# B&R Automation Studio project TD52 (part 50)

#### perm_par.var
```iecst
VAR
	tParaIntern : ParaHandler_typ; (*Connector type to perm_par*)
	tMM2ParaBase_ReadBack : MM2ParaBase_type; (*INTERNAL! V4.06 new readback structure for information from previous tasks*)
	bWriteDataObj : BOOL; (* TRUE=write data object module *)
	bDataObjLenErr : BOOL; (*Error occured in permem: data module size missmatch*)
	bCreateDataObj : BOOL; (* TRUE=create new data object *)
	bWriteOnce : BOOL; (* write permanent memory once *)
	DatObjCreate_01 : DatObjCreate; (* data object create *)
	DatObjInfoBak_02 : DatObjInfo; (* data object info *)
	DatObjDelete_01 : DatObjDelete; (* data object delete *)
	DatObjRead_01 : DatObjRead; (* data object read *)
	DatObjRead_02 : DatObjRead; (* manual initiated data object read *)
	DatObjWrite_01 : DatObjWrite; (* data object write *)
	DatObjDelete_02 : DatObjDelete; (* data object delete *)
	DatObjDelete_11 : DatObjDelete; (*Delete Backup File*)
	DatObjInfo_01 : DatObjInfo; (* data object info *)
	DatObjInfo_02 : DatObjInfo; (* data object info *)
	szModuleName : STRING[35]; (* module name of object *)
	szModuleNameBackup : STRING[35]; (* module name of posiibly created backup object *)
	DatObjCopy_01 : DatObjCopy;
	bCopyDataObj : BOOL;
	TON_WarnDelay : TON;
	TON_WritePMEM : TON; (* delay write permanent memory *)
	ulPMPointer : UDINT; (* adress of actual checksum value *)
	ulChecksum : UDINT; (* parameter checksum value *)
	pm_len : UDINT; (* permanent value lenght *)
	ulChecksumOld : UDINT; (* last vlaue of parameter checksum *)
	ulChkValue : UDINT; (* actual value of parameter pointer *)
	pm_id : UDINT; (* permanent value identifier *)
	pm_p : UDINT; (* permanent value pointer *)
	DatObjInfo_META : DatObjInfo;
	DatObjRead_META : DatObjRead;
	szMetaDataRaw : STRING[2000];
	szMetaData : ARRAY[0..4] OF STRING[35];
	szMetaDataVis : ARRAY[0..3] OF STRING[35];
	ssIndex : INT;
	ssCount : INT;
	ucMetaDataRaw : ARRAY[0..2000] OF USINT;
	ssCount2 : INT;
	szMetaDataFile : STRING[10];
	szText1 : STRING[20];
	pv_adr_IN_XX_tPB2MM : UDINT;
	pv_lng : UDINT;
	pv_lng_IN_XX_tPB2MM : UDINT;
	pv_lng_OUT_XX_tPB2MM : UDINT;
	szText2 : STRING[20];
	pv_adr_OUT_XX_tXX2PB : UDINT;
END_VAR
VAR CONSTANT
	ERR_NOERROR : UINT := 0;
END_VAR
VAR
	usPMWriteCnt : UINT;
	pm_Error : UDINT; (* permanent value error *) (* Deleted: pm : ParaMem_typ; permanent memory tags mathias, 22.8.11*)
	fun_Error : UDINT := 0; (*state > 0 = function error*)
	xLocalParaCheck : ParaCheckFUB; (*local function instance to check parameter values*)
	TON_ParaSetupOk : TON;
	bParaCheckSystemOk : BOOL;
	iDebug_ParaOkChecked : UDINT;
	bRestoreBackupDataObj : BOOL := FALSE;
	bRestoreDataObjContent : BOOL := FALSE;
	pm_id_backup : UDINT;
	pm_p_Backup : UDINT;
	DatObjCopy_02 : DatObjCopy;
	bDeleteBackupDataObj : BOOL := FALSE; (*Command to delete backup data module file on purpose*)
	bDebugPara : ARRAY[0..5] OF BOOL;
	ssIndex2 : INT;
	ssIndex3 : INT;
	ssIndex4 : INT;
	ssIndexVis : INT;
	szText : STRING[40];
	pv_adr_Para : UDINT;
	szParaSnippet : ARRAY[0..5] OF STRING[150];
	szParaIndex : STRING[10];
	slValue : DINT;
	iModuleDLD_ResetCount : INT;
	bDownloadDetected : BOOL;
	bFlagParaStructCopyWorking : BOOL; (*true, if cyclic para copying is active, 1 false cycle at every copy *)
	bStoreInitParaInDataObj : BOOL := FALSE;
	bTestflag : BOOL;
	bReadOutMETA_Once : BOOL;
	tParaCheck_iPvAdress : ARRAY[0..5] OF UDINT;
	tParaCheck_iPvLengt : ARRAY[0..5] OF UDINT;
	tParaCheck_rPvValue : ARRAY[0..5] OF REAL;
	tParaCheck_rRangeMIN : ARRAY[0..5] OF REAL;
	tParaCheck_rRangeMAX : ARRAY[0..5] OF REAL;
	tParaCheck_szPvName : ARRAY[0..5] OF STRING[35];
	ssFormatDetected : INT;
	szMetaDataPart : STRING[150];
	szFullTaskName : STRING[35];
	szFullMetaModuleName : STRING[35];
	debugLen : INT;
	debugSize : INT := 0;
	strcat_adr1 : UDINT;
	strcat_adr2 : UDINT;
	ssIndexTN : INT;
	bAlternate : BOOL;
	n : INT;
	iAlternateChecksum : DINT;
	iAlternateChecksumOld : DINT;
	ulDebugChkValue : ARRAY[0..999] OF UDINT;
	Adr1 : UDINT;
	Adr2 : UDINT;
	usPMWriteCntStepsize : UINT := 1; (*different step sizes to help debug*)
	usPMWriteCntXOR : UINT;
	usPMWriteCntAltSum : UINT;
	ulAdrPM : UDINT;
	usChkValuePM : USINT;
	ulAdrPara : UDINT;
	ulPara_len : UDINT;
	usChkValuePara : USINT;
	iDebugCountPMDifferences : DINT := 0;
	bEngineRunDetected : BOOL; (*detection status bit autocommand 100 /101  for engine run state*)
	ucMetaDataDebugInfoLine : ARRAY[0..24] OF STRING[80];
	ssIndexMand : INT := 0;
	szMetaDataMand : STRING[35];
	iMyErrorInfo_Autoreset : DINT; (*internal autoreset counter*)
	ssIndex_Version : INT; (*internal*)
	ssIndex_BU : INT; (*internal*)
	ssIndex_BU2 : INT; (*internal*)
END_VAR
```

### Program Logical/Customized/Cust_Internals/par_UniFile (IEC, version 0.99.0) - + obsolete

- par_UniFile.st (not readable text: treated as protected, skipped)

### Program Logical/Customized/Cust_Internals/par_UniString (IEC, version 1.06.0) - + obsolete

- par_UniString.st (not readable text: treated as protected, skipped)

### Program Logical/Customized/Cust_Internals/par_Universal_IO (IEC, version 1.16.0) - + obsolete

- par_Universal_IO.st (not readable text: treated as protected, skipped)

### Program Logical/Customized/Cust_Internals/MsgCUInternal (IEC, version 4.10.0) - + unchangeable module messages

- MsgCUInterCyclic.st (not readable text: treated as protected, skipped)

- MsgCUInterInit.st (not readable text: treated as protected, skipped)

#### MsgCUInter.var - Local variables
```iecst
(********************************************************************
 * COPYRIGHT -- INNIO Company
 ********************************************************************
 * Program: MsgCUInter
 * File: MsgCUInter.var
 * Author: zengerer
 * Created: September 10, 2013
 ********************************************************************
 * Local variables of program MsgCU
 ********************************************************************)
VAR
	iAdrAmmBase2MM : UDINT;
	iAdrMM2AmmBase : UDINT;
	xMsg13 : ARRAY[0..99] OF Msg; (*Array of Msg for Reserve Analog IN*)
	xMsg14 : ARRAY[0..99] OF Msg; (*Array of Msg for Reserve Analog IN*)
	xMsg1500 : Msg; (*Msg 1500 for Reserve Analog IN*)
	xMsg37 : ARRAY[0..99] OF Msg; (*Array of Msg for Reserve Analog IN*)
	xMsg38 : ARRAY[0..99] OF Msg; (*Array of Msg for Reserve Analog IN*)
	xMsg39 : ARRAY[0..99] OF Msg; (*Array of Msg for Reserve Analog IN*)
	xMsg89 : ARRAY[66..99] OF Msg; (*Array of Msg for CustomerIO and Reserve AI*)
END_VAR
```

### Program Logical/Customized/Cust_Internals/ran_Internal (IEC, version 4.12.0) - + processing of spare analog inputs,..

- ran_InternalCyclic.st (not readable text: treated as protected, skipped)

#### ran_Internal.var
```iecst
VAR
	xTON_lim_LoLo : ARRAY[0..120] OF TON;
	xTON_lim_lo : ARRAY[0..120] OF TON;
	xTON_lim_hi : ARRAY[0..120] OF TON;
	xTON_lim_HiHi : ARRAY[0..120] OF TON;
	xLCRScal_10 : LCRScal;
	xLCRScal_15 : LCRScal;
	xLCRScal_16 : LCRScal;
	bGR_MIN_lim_LoLo_Q : BOOL := 0;
	bGR_MIN_lim_lo_Q : BOOL := 0;
	bGR_MAX_lim_hi_Q : BOOL := 0;
	bGR_MAX_lim_HiHi_Q : BOOL := 0;
END_VAR
```

### Data object Logical/Customized/aeprot (Simple, version 4.01.0) - modification report

#### aeprot.dat
```
; modification report
;----------------------------------------------------------------------
 "<BASEVERSION>04.25.00.00</BASEVERSION>"   ;	(XT4) | 05.02.2026
; (The version number above is unchangeable, except for basic software releases. Do NOT change for any customizations, which have to get versioned in the META modules!)
;
; Bugs&Solutions		       :  V.. / xx.xx.202x / ..
;
; update                  :  .... / xx.xx.202x / ..
;
; VSoftworker             :  1.1.9.4
;
; cross reference for DIA.NE VIS
;  - reserve failures used     : Y/N  : ..
;  - reserve controllers       : Y/N
;  - reserve operation messages: Y/N  : ..
;  - change of main loop       : Y/N  : ..
;
; customer-specifics
;  - standard of               :  ..
;  - auxiliary controls        :  Y/N
;
; copy
;  - derived from              :  J....
;  - copied 1:1                :  N
;
; new version                   :  04.25.00.01
; date of design          		:  10.02.2026
; author                  		:  Nuschele Lukas
;
;
; module                       : HalIO
; task                         : IOcfg
; modification                 : Block T_GT_NG | Type | von AI_0_20mA_INT16 auf AI_TEMP_1_10C geändert
;											   | Qual_Min | von 4914 auf -200 geändert
;											   | Qual_Max | von 32767 auf 1400 geändert
;											   | Scal_X1 | von 6552 auf 0 geändert
;											   | Scal_X2 | von 32760 auf 0 geändert
;
; reason for modification      : ist kein mA Signal sondern ein PT100
;
;
; WinMOD tested				   : Y/N
;
; new version                  :  04.25.00.02
; date of design          	   :  11.02.2026
; author               	       :  Bacci
;
; META version changed         :  Y "<VERSION>04.24.00.03</VERSION>"
; module 			           :  EngineGeneral
; task                         :  VibMonEG, VibMon2EG, VibMon3EG
; modification                 :  vibration sensors 5 - 12 added
;
; reason for modification      :  additional vibration sensors needed, customized for DP29
;
;
; new version                  :  04.25.00.03
; date of design          	   :  25.03.2026
; author               	       :  Vockenberger
;
; changed DP29 to DT52
; INFO for jenbacher test bench	: 	DCGA will be put into operation later with the V4.26 release.
;									P29 (according to the wiring diagram) will be put into operation later by the development team.
;
;----------------------------------------------------------------------
; jenbacher test bench
;
; new version                  :  04.25.00.02
;
; check date     (TPE)         :  xx.xx.202x
; checked from   (TPE)         :  ..
; start-up without
; source-code    (TPE)    	   :  Y/N
;
;----------------------------------------------------------------------
;
; softw.instal.(pre-testbench) :  xx.xx.202x
; installed by (pre-testbench) :  ..
; modifications			       :  Y/N
;
; date of modification         :  xx.xx.202x
; modified by                  :
;
;
; META version changed         :  Y/N
; module                       :
; task                         :
; modification                 :
;
; reason for modification      :
;
;----------------------------------------------------------------------
;
; softw.instal.(unit-testbench):  xx.xx.2026
; installed by (unit-testbench):
; modifications			       :  Y/N
;
; date of modification         :
; modified by                  :
;
;
; META version changed         :  Y/N
; module                       :
; task                         :
; modification                 :
;
; reason for modification      :
;
; META version changed         :  Y/N
; module                       :
; task                         :
; modification                 :
;
; reason for modification      :
;
;----------------------------------------------------------------------
; start-up
;
; softw.install. (Service)     :  xx.xx.202x
; installed by   (Service)     :  ..
; check date     (TPE)         :  xx.xx.202x
; checked from   (TPE)         :  ..
;
"*********************************************************************"
"                                                                     "
"! ! ! ! ! ! !   please update version info in META_CU  ! ! ! ! ! ! ! "
"                                                                     "
"*********************************************************************"
; new version                  :  04.25.00.03
;
; date of modif. (TPE)         :  12.03.2026
; modified by    (TPE)         :  Bencze
; softw.install. (Service)     :  xx.xx.202x
; installed by   (Service)     :  ..
;
; date of modif. (Service)     :  xx.xx.202x
; modified by    (Service)     :  ..
; check date     (TPE)         :  xx.xx.202x
; checked from   (TPE)         :  ..
;
; META version changed         :  Y
; module                       :  CU
; task                         :  c_clutch_CAN
; modification                 :  CAN values integration

; META version changed         :  Y
; module                       :  CU
; task                         :  MsgCU
; modification                 :  W1756 to W1765
;
; reason for modification      : Working Clutch setup
;
"*********************************************************************"
"                                                                     "
"! ! ! ! ! ! !   please update version info in META_CU  ! ! ! ! ! ! ! "
"                                                                     "
"*********************************************************************"
; new version                  :  04.25.00.xx
;
; date of modif. (TPE)         :  xx.xx.202x
; modified by    (TPE)         :  ..
; softw.install. (Service)     :  xx.xx.202x
; installed by   (Service)     :  ..
;
; date of modif. (Service)     :  xx.xx.202x
; modified by    (Service)     :  ..
; check date     (TPE)         :  xx.xx.202x
; checked from   (TPE)         :  ..
;
; META version changed         :  Y/N
; module                       :
; task                         :
; modification                 :
;
; reason for modification      :
;
"*********************************************************************"
"                                                                     "
"! ! ! ! ! ! !   please update version info in META_CU  ! ! ! ! ! ! ! "
"                                                                     "
"*********************************************************************"
; new version                  :  04.25.00.xx
;
; date of modif. (TPE)         :  xx.xx.202x
; modified by    (TPE)         :  ..
; softw.install. (Service)     :  xx.xx.202x
; installed by   (Service)     :  ..
;
; date of modif. (Service)     :  xx.xx.202x
; modified by    (Service)     :  ..
; check date     (TPE)         :  xx.xx.202x
; checked from   (TPE)         :  ..
;
; META version changed         :  Y/N
; module                       :
; task                         :
; modification                 :
;
; reason for modification      :
;
"*********************************************************************"
"                                                                     "
"! ! ! ! ! ! !   please update version info in META_CU  ! ! ! ! ! ! ! "
"                                                                     "
"*********************************************************************"
; new version                  :  04.25.00.xx
;
; date of modif. (TPE)         :  xx.xx.202x
; modified by    (TPE)         :  ..
; softw.install. (Service)     :  xx.xx.202x
; installed by   (Service)     :  ..
;
; date of modif. (Service)     :  xx.xx.202x
; modified by    (Service)     :  ..
; check date     (TPE)         :  xx.xx.202x
; checked from   (TPE)         :  ..
;
; META version changed         :  Y/N
; module                       :
; task                         :
; modification                 :
;
; reason for modification      :
;
"*********************************************************************"
"                                                                     "
"! ! ! ! ! ! !   please update version info in META_CU  ! ! ! ! ! ! ! "
"                                                                     "
"*********************************************************************"
; new version                  :  04.25.00.xx
;
; date of modif. (TPE)         :  xx.xx.202x
; modified by    (TPE)         :  ..
; softw.install. (Service)     :  xx.xx.202x
; installed by   (Service)     :  ..
;
; date of modif. (Service)     :  xx.xx.202x
; modified by    (Service)     :  ..
; check date     (TPE)         :  xx.xx.202x
; checked from   (TPE)         :  ..
;
; META version changed         :  Y/N
; module                       :
; task                         :
; modification                 :
;
; reason for modification      :
;
```

### Program Logical/Customized/PlantCom/c_PlantComMap10ms (IEC, version 4.14.0)

#### Cyclic.st - Cyclic code
```iecst
(*******************************************************************************
Customized Variable mapping for the plant communication

This code is confidential and proprietary to the INNIO Company.
It may not be used in any form, or reproduced in any manner, without the express
written permission of the INNIO Company.
Copyright, INNIO Company, 2024

Customized modifications: -
------------------------

History:
-------
V4.14.0	26.11.2024	Astner	Created Task

Instructions for use:
--------------------
Replace the bPlaceholderCustomSignal[x] variable with the variable you want to add to the plant communication.
The GoodQual Value of the Output variables must be always true by default, if additional logic is needed this
has to be implemented in the software module where the variable is coming from.
The GoodQual Value of the inputs is set by the communication participant.

Outstandings:
------------

*******************************************************************************)
PROGRAM _CYCLIC
	(* Do not exeucte mapping if plant communication is not configured *)
	IF (NOT IN_CU.bPlantComCfgOk) THEN
		RETURN;
	END_IF
	(***************************************************)
	(*** Customized Inputs from the master controls  ***)
	(***************************************************)
	FOR x:=Para.tPlantComm.iMas_Num_Min TO Para.tPlantComm.iMas_Num_Max DO
		(***********************)
		(*** Digital Signals ***)
		(***********************)

		(* Reserve Signal 1 *)
		bPlaceHolderCustomSignal[x] 			:= IN_CU.tPlantCom_M2E_In_Cust10ms[x].digitalSignals[digOffset+80].Value;
		bPlaceHolderCustomSignalGoodQual[x] 	:= IN_CU.tPlantCom_M2E_In_Cust10ms[x].digitalSignals[digOffset+80].GoodQual;

		(* Reserve Signal 2 *)
		bPlaceHolderCustomSignal[x] 			:= IN_CU.tPlantCom_M2E_In_Cust10ms[x].digitalSignals[digOffset+81].Value;
		bPlaceHolderCustomSignalGoodQual[x] 	:= IN_CU.tPlantCom_M2E_In_Cust10ms[x].digitalSignals[digOffset+81].GoodQual;

		(* Reserve Signal 3 *)
		bPlaceHolderCustomSignal[x] 			:= IN_CU.tPlantCom_M2E_In_Cust10ms[x].digitalSignals[digOffset+82].Value;
		bPlaceHolderCustomSignalGoodQual[x] 	:= IN_CU.tPlantCom_M2E_In_Cust10ms[x].digitalSignals[digOffset+82].GoodQual;

		(* Reserve Signal 4 *)
		bPlaceHolderCustomSignal[x] 			:= IN_CU.tPlantCom_M2E_In_Cust10ms[x].digitalSignals[digOffset+83].Value;
		bPlaceHolderCustomSignalGoodQual[x] 	:= IN_CU.tPlantCom_M2E_In_Cust10ms[x].digitalSignals[digOffset+83].GoodQual;

		(* Reserve Signal 5 *)
		bPlaceHolderCustomSignal[x] 			:= IN_CU.tPlantCom_M2E_In_Cust10ms[x].digitalSignals[digOffset+84].Value;
		bPlaceHolderCustomSignalGoodQual[x] 	:= IN_CU.tPlantCom_M2E_In_Cust10ms[x].digitalSignals[digOffset+84].GoodQual;

		(* Reserve Signal 6 *)
		bPlaceHolderCustomSignal[x]				:= IN_CU.tPlantCom_M2E_In_Cust10ms[x].digitalSignals[digOffset+85].Value;
		bPlaceHolderCustomSignalGoodQual[x] 	:= IN_CU.tPlantCom_M2E_In_Cust10ms[x].digitalSignals[digOffset+85].GoodQual;

		(* Reserve Signal 7 *)
		bPlaceHolderCustomSignal[x] 			:= IN_CU.tPlantCom_M2E_In_Cust10ms[x].digitalSignals[digOffset+86].Value;
		bPlaceHolderCustomSignalGoodQual[x] 	:= IN_CU.tPlantCom_M2E_In_Cust10ms[x].digitalSignals[digOffset+86].GoodQual;

		(* Reserve Signal 8 *)
		bPlaceHolderCustomSignal[x] 			:= IN_CU.tPlantCom_M2E_In_Cust10ms[x].digitalSignals[digOffset+87].Value;
		bPlaceHolderCustomSignalGoodQual[x] 	:= IN_CU.tPlantCom_M2E_In_Cust10ms[x].digitalSignals[digOffset+87].GoodQual;

		(* Reserve Signal 9 *)
		bPlaceHolderCustomSignal[x] 			:= IN_CU.tPlantCom_M2E_In_Cust10ms[x].digitalSignals[digOffset+88].Value;
		bPlaceHolderCustomSignalGoodQual[x] 	:= IN_CU.tPlantCom_M2E_In_Cust10ms[x].digitalSignals[digOffset+88].GoodQual;

		(* Reserve Signal 10 *)
		bPlaceHolderCustomSignal[x] 			:= IN_CU.tPlantCom_M2E_In_Cust10ms[x].digitalSignals[digOffset+89].Value;
		bPlaceHolderCustomSignalGoodQual[x] 	:= IN_CU.tPlantCom_M2E_In_Cust10ms[x].digitalSignals[digOffset+89].GoodQual;

		(* Reserve Signal 11 *)
		bPlaceHolderCustomSignal[x] 			:= IN_CU.tPlantCom_M2E_In_Cust10ms[x].digitalSignals[digOffset+90].Value;
		bPlaceHolderCustomSignalGoodQual[x] 	:= IN_CU.tPlantCom_M2E_In_Cust10ms[x].digitalSignals[digOffset+90].GoodQual;

		(* Reserve Signal 12 *)
		bPlaceHolderCustomSignal[x] 			:= IN_CU.tPlantCom_M2E_In_Cust10ms[x].digitalSignals[digOffset+91].Value;
		bPlaceHolderCustomSignalGoodQual[x] 	:= IN_CU.tPlantCom_M2E_In_Cust10ms[x].digitalSignals[digOffset+91].GoodQual;

		(* Reserve Signal 13 *)
		bPlaceHolderCustomSignal[x] 			:= IN_CU.tPlantCom_M2E_In_Cust10ms[x].digitalSignals[digOffset+92].Value;
		bPlaceHolderCustomSignalGoodQual[x] 	:= IN_CU.tPlantCom_M2E_In_Cust10ms[x].digitalSignals[digOffset+92].GoodQual;

		(* Reserve Signal 14 *)
		bPlaceHolderCustomSignal[x] 			:= IN_CU.tPlantCom_M2E_In_Cust10ms[x].digitalSignals[digOffset+93].Value;
		bPlaceHolderCustomSignalGoodQual[x] 	:= IN_CU.tPlantCom_M2E_In_Cust10ms[x].digitalSignals[digOffset+93].GoodQual;

		(* Reserve Signal 15 *)
		bPlaceHolderCustomSignal[x] 			:= IN_CU.tPlantCom_M2E_In_Cust10ms[x].digitalSignals[digOffset+94].Value;
		bPlaceHolderCustomSignalGoodQual[x] 	:= IN_CU.tPlantCom_M2E_In_Cust10ms[x].digitalSignals[digOffset+94].GoodQual;

		(* Reserve Signal 16 *)
		bPlaceHolderCustomSignal[x] 			:= IN_CU.tPlantCom_M2E_In_Cust10ms[x].digitalSignals[digOffset+95].Value;
		bPlaceHolderCustomSignalGoodQual[x] 	:= IN_CU.tPlantCom_M2E_In_Cust10ms[x].digitalSignals[digOffset+95].GoodQual;

		(**********************)
		(*** Analog Signals ***)
		(**********************)

		(* Reserve Signal 1 *)
		rPlaceHolderCustomSignal[x] 			:= IN_CU.tPlantCom_M2E_In_Cust10ms[x].analogSignals[anaOffset+40].Value;
		bPlaceHolderCustomSignalGoodQual[x] 	:= IN_CU.tPlantCom_M2E_In_Cust10ms[x].analogSignals[anaOffset+40].GoodQual;

		(* Reserve Signal 2 *)
		rPlaceHolderCustomSignal[x] 			:= IN_CU.tPlantCom_M2E_In_Cust10ms[x].analogSignals[anaOffset+41].Value;
		bPlaceHolderCustomSignalGoodQual[x] 	:= IN_CU.tPlantCom_M2E_In_Cust10ms[x].analogSignals[anaOffset+41].GoodQual;

		(* Reserve Signal 3 *)
		rPlaceHolderCustomSignal[x] 			:= IN_CU.tPlantCom_M2E_In_Cust10ms[x].analogSignals[anaOffset+42].Value;
		bPlaceHolderCustomSignalGoodQual[x] 	:= IN_CU.tPlantCom_M2E_In_Cust10ms[x].analogSignals[anaOffset+42].GoodQual;

		(* Reserve Signal 4 *)
		rPlaceHolderCustomSignal[x] 			:= IN_CU.tPlantCom_M2E_In_Cust10ms[x].analogSignals[anaOffset+43].Value;
		bPlaceHolderCustomSignalGoodQual[x] 	:= IN_CU.tPlantCom_M2E_In_Cust10ms[x].analogSignals[anaOffset+43].GoodQual;

		(* Reserve Signal 5 *)
		rPlaceHolderCustomSignal[x] 			:= IN_CU.tPlantCom_M2E_In_Cust10ms[x].analogSignals[anaOffset+44].Value;
		bPlaceHolderCustomSignalGoodQual[x] 	:= IN_CU.tPlantCom_M2E_In_Cust10ms[x].analogSignals[anaOffset+44].GoodQual;

		(* Reserve Signal 6 *)
		rPlaceHolderCustomSignal[x]	 			:= IN_CU.tPlantCom_M2E_In_Cust10ms[x].analogSignals[anaOffset+45].Value;
		bPlaceHolderCustomSignalGoodQual[x] 	:= IN_CU.tPlantCom_M2E_In_Cust10ms[x].analogSignals[anaOffset+45].GoodQual;

		(* Reserve Signal 7 *)
		rPlaceHolderCustomSignal[x] 			:= IN_CU.tPlantCom_M2E_In_Cust10ms[x].analogSignals[anaOffset+46].Value;
		bPlaceHolderCustomSignalGoodQual[x] 	:= IN_CU.tPlantCom_M2E_In_Cust10ms[x].analogSignals[anaOffset+46].GoodQual;

		(* Reserve Signal 8 *)
		rPlaceHolderCustomSignal[x] 			:= IN_CU.tPlantCom_M2E_In_Cust10ms[x].analogSignals[anaOffset+47].Value;
		bPlaceHolderCustomSignalGoodQual[x] 	:= IN_CU.tPlantCom_M2E_In_Cust10ms[x].analogSignals[anaOffset+47].GoodQual;
	END_FOR

	(*** Customized Outputs to the master controls  ***)
	FOR x:=Para.tPlantComm.iMas_Num_Min TO Para.tPlantComm.iMas_Num_Max DO
		(***********************)
		(*** Digital Signals ***)
		(***********************)
		bPlaceHolderCustomSignal[x] := FALSE;
		(* Reserve Signal 1 *)
		OUT_CU.tPlantCom_E2M_Out_Cust10ms[x].digitalSignals[digOffset+80].Value 		:= bPlaceHolderCustomSignal[x];
		OUT_CU.tPlantCom_E2M_Out_Cust10ms[x].digitalSignals[digOffset+80].GoodQual		:= TRUE;

		(* Reserve Signal 2 *)
		OUT_CU.tPlantCom_E2M_Out_Cust10ms[x].digitalSignals[digOffset+81].Value 		:= bPlaceHolderCustomSignal[x];
		OUT_CU.tPlantCom_E2M_Out_Cust10ms[x].digitalSignals[digOffset+81].GoodQual		:= TRUE;

		(* Reserve Signal 3 *)
		OUT_CU.tPlantCom_E2M_Out_Cust10ms[x].digitalSignals[digOffset+82].Value 		:= bPlaceHolderCustomSignal[x];
		OUT_CU.tPlantCom_E2M_Out_Cust10ms[x].digitalSignals[digOffset+82].GoodQual		:= TRUE;

		(* Reserve Signal 4 *)
		OUT_CU.tPlantCom_E2M_Out_Cust10ms[x].digitalSignals[digOffset+83].Value 		:= bPlaceHolderCustomSignal[x];
		OUT_CU.tPlantCom_E2M_Out_Cust10ms[x].digitalSignals[digOffset+83].GoodQual		:= TRUE;

		(* Reserve Signal 5 *)
		OUT_CU.tPlantCom_E2M_Out_Cust10ms[x].digitalSignals[digOffset+84].Value 		:= bPlaceHolderCustomSignal[x];
		OUT_CU.tPlantCom_E2M_Out_Cust10ms[x].digitalSignals[digOffset+84].GoodQual		:= TRUE;

		(* Reserve Signal 6 *)
		OUT_CU.tPlantCom_E2M_Out_Cust10ms[x].digitalSignals[digOffset+85].Value 		:= bPlaceHolderCustomSignal[x];
		OUT_CU.tPlantCom_E2M_Out_Cust10ms[x].digitalSignals[digOffset+85].GoodQual		:= TRUE;

		(* Reserve Signal 7 *)
		OUT_CU.tPlantCom_E2M_Out_Cust10ms[x].digitalSignals[digOffset+86].Value			:= bPlaceHolderCustomSignal[x];
		OUT_CU.tPlantCom_E2M_Out_Cust10ms[x].digitalSignals[digOffset+86].GoodQual		:= TRUE;

		(* Reserve Signal 8 *)
		OUT_CU.tPlantCom_E2M_Out_Cust10ms[x].digitalSignals[digOffset+87].Value 		:= bPlaceHolderCustomSignal[x];
		OUT_CU.tPlantCom_E2M_Out_Cust10ms[x].digitalSignals[digOffset+87].GoodQual		:= TRUE;

		(* Reserve Signal 9 *)
		OUT_CU.tPlantCom_E2M_Out_Cust10ms[x].digitalSignals[digOffset+88].Value 		:= bPlaceHolderCustomSignal[x];
		OUT_CU.tPlantCom_E2M_Out_Cust10ms[x].digitalSignals[digOffset+88].GoodQual		:= TRUE;

		(* Reserve Signal 10 *)
		OUT_CU.tPlantCom_E2M_Out_Cust10ms[x].digitalSignals[digOffset+89].Value 		:= bPlaceHolderCustomSignal[x];
		OUT_CU.tPlantCom_E2M_Out_Cust10ms[x].digitalSignals[digOffset+89].GoodQual		:= TRUE;

		(* Reserve Signal 11 *)
		OUT_CU.tPlantCom_E2M_Out_Cust10ms[x].digitalSignals[digOffset+90].Value 		:= bPlaceHolderCustomSignal[x];
		OUT_CU.tPlantCom_E2M_Out_Cust10ms[x].digitalSignals[digOffset+90].GoodQual		:= TRUE;

		(* Reserve Signal 12 *)
		OUT_CU.tPlantCom_E2M_Out_Cust10ms[x].digitalSignals[digOffset+91].Value 		:= bPlaceHolderCustomSignal[x];
		OUT_CU.tPlantCom_E2M_Out_Cust10ms[x].digitalSignals[digOffset+91].GoodQual		:= TRUE;

		(* Reserve Signal 13 *)
		OUT_CU.tPlantCom_E2M_Out_Cust10ms[x].digitalSignals[digOffset+92].Value 		:= bPlaceHolderCustomSignal[x];
		OUT_CU.tPlantCom_E2M_Out_Cust10ms[x].digitalSignals[digOffset+92].GoodQual		:= TRUE;

		(* Reserve Signal 14 *)
		OUT_CU.tPlantCom_E2M_Out_Cust10ms[x].digitalSignals[digOffset+93].Value 		:= bPlaceHolderCustomSignal[x];
		OUT_CU.tPlantCom_E2M_Out_Cust10ms[x].digitalSignals[digOffset+93].GoodQual		:= TRUE;

		(* Reserve Signal 15 *)
		OUT_CU.tPlantCom_E2M_Out_Cust10ms[x].digitalSignals[digOffset+94].Value 		:= bPlaceHolderCustomSignal[x];
		OUT_CU.tPlantCom_E2M_Out_Cust10ms[x].digitalSignals[digOffset+94].GoodQual		:= TRUE;

		(* Reserve Signal 16 *)
		OUT_CU.tPlantCom_E2M_Out_Cust10ms[x].digitalSignals[digOffset+95].Value 		:= bPlaceHolderCustomSignal[x];
		OUT_CU.tPlantCom_E2M_Out_Cust10ms[x].digitalSignals[digOffset+95].GoodQual		:= TRUE;

		(**********************)
		(*** Analog Signals ***)
		(**********************)
		rPlaceHolderCustomSignal[x] := 0.0;
		(* Reserve Signal 1 *)
		OUT_CU.tPlantCom_E2M_Out_Cust10ms[x].analogSignals[anaOffset+40].Value 		:= rPlaceHolderCustomSignal[x];
		OUT_CU.tPlantCom_E2M_Out_Cust10ms[x].analogSignals[anaOffset+40].GoodQual	:= TRUE;

		(* Reserve Signal 2 *)
		OUT_CU.tPlantCom_E2M_Out_Cust10ms[x].analogSignals[anaOffset+41].Value 		:= rPlaceHolderCustomSignal[x];
		OUT_CU.tPlantCom_E2M_Out_Cust10ms[x].analogSignals[anaOffset+41].GoodQual	:= TRUE;

		(* Reserve Signal 3 *)
		OUT_CU.tPlantCom_E2M_Out_Cust10ms[x].analogSignals[anaOffset+42].Value 		:= rPlaceHolderCustomSignal[x];
		OUT_CU.tPlantCom_E2M_Out_Cust10ms[x].analogSignals[anaOffset+42].GoodQual	:= TRUE;

		(* Reserve Signal 4 *)
		OUT_CU.tPlantCom_E2M_Out_Cust10ms[x].analogSignals[anaOffset+43].Value 		:= rPlaceHolderCustomSignal[x];
		OUT_CU.tPlantCom_E2M_Out_Cust10ms[x].analogSignals[anaOffset+43].GoodQual	:= TRUE;

		(* Reserve Signal 5 *)
		OUT_CU.tPlantCom_E2M_Out_Cust10ms[x].analogSignals[anaOffset+44].Value 		:= rPlaceHolderCustomSignal[x];
		OUT_CU.tPlantCom_E2M_Out_Cust10ms[x].analogSignals[anaOffset+44].GoodQual	:= TRUE;

		(* Reserve Signal 6 *)
		OUT_CU.tPlantCom_E2M_Out_Cust10ms[x].analogSignals[anaOffset+45].Value 		:= rPlaceHolderCustomSignal[x];
		OUT_CU.tPlantCom_E2M_Out_Cust10ms[x].analogSignals[anaOffset+45].GoodQual	:= TRUE;

		(* Reserve Signal 7 *)
		OUT_CU.tPlantCom_E2M_Out_Cust10ms[x].analogSignals[anaOffset+46].Value 		:= rPlaceHolderCustomSignal[x];
		OUT_CU.tPlantCom_E2M_Out_Cust10ms[x].analogSignals[anaOffset+46].GoodQual	:= TRUE;

		(* Reserve Signal 8 *)
		OUT_CU.tPlantCom_E2M_Out_Cust10ms[x].analogSignals[anaOffset+47].Value 		:= rPlaceHolderCustomSignal[x];
		OUT_CU.tPlantCom_E2M_Out_Cust10ms[x].analogSignals[anaOffset+47].GoodQual	:= TRUE;
	END_FOR

	(*** Customized Inputs from the other engines ***)
	FOR x:=Para.tPlantComm.iEng_Num_Min TO Para.tPlantComm.iEng_Num_Max DO
		(***********************)
		(*** Digital Signals ***)
		(***********************)

		(* Reserve Signal 1 *)
		bPlaceHolderCustomSignal[x] 				:= IN_CU.tPlantCom_E2E_In_Cust10ms[x].digitalSignals[digOffset+80].Value;
		bPlaceHolderCustomSignalGoodQual[x] 		:= IN_CU.tPlantCom_E2E_In_Cust10ms[x].digitalSignals[digOffset+80].GoodQual;

		(* Reserve Signal 2 *)
		bPlaceHolderCustomSignal[x] 				:= IN_CU.tPlantCom_E2E_In_Cust10ms[x].digitalSignals[digOffset+81].Value;
		bPlaceHolderCustomSignalGoodQual[x] 		:= IN_CU.tPlantCom_E2E_In_Cust10ms[x].digitalSignals[digOffset+81].GoodQual;

		(* Reserve Signal 3 *)
		bPlaceHolderCustomSignal[x] 				:= IN_CU.tPlantCom_E2E_In_Cust10ms[x].digitalSignals[digOffset+82].Value;
		bPlaceHolderCustomSignalGoodQual[x] 		:= IN_CU.tPlantCom_E2E_In_Cust10ms[x].digitalSignals[digOffset+82].GoodQual;

		(* Reserve Signal 4 *)
		bPlaceHolderCustomSignal[x] 				:= IN_CU.tPlantCom_E2E_In_Cust10ms[x].digitalSignals[digOffset+83].Value;
		bPlaceHolderCustomSignalGoodQual[x] 		:= IN_CU.tPlantCom_E2E_In_Cust10ms[x].digitalSignals[digOffset+83].GoodQual;

		(* Reserve Signal 5 *)
		bPlaceHolderCustomSignal[x] 				:= IN_CU.tPlantCom_E2E_In_Cust10ms[x].digitalSignals[digOffset+84].Value;
		bPlaceHolderCustomSignalGoodQual[x] 		:= IN_CU.tPlantCom_E2E_In_Cust10ms[x].digitalSignals[digOffset+84].GoodQual;

		(* Reserve Signal 6 *)
		bPlaceHolderCustomSignal[x] 				:= IN_CU.tPlantCom_E2E_In_Cust10ms[x].digitalSignals[digOffset+85].Value;
		bPlaceHolderCustomSignalGoodQual[x] 		:= IN_CU.tPlantCom_E2E_In_Cust10ms[x].digitalSignals[digOffset+85].GoodQual;

		(* Reserve Signal 7 *)
		bPlaceHolderCustomSignal[x] 				:= IN_CU.tPlantCom_E2E_In_Cust10ms[x].digitalSignals[digOffset+86].Value;
		bPlaceHolderCustomSignalGoodQual[x] 		:= IN_CU.tPlantCom_E2E_In_Cust10ms[x].digitalSignals[digOffset+86].GoodQual;

		(* Reserve Signal 8 *)
		bPlaceHolderCustomSignal[x] 				:= IN_CU.tPlantCom_E2E_In_Cust10ms[x].digitalSignals[digOffset+87].Value;
		bPlaceHolderCustomSignalGoodQual[x] 		:= IN_CU.tPlantCom_E2E_In_Cust10ms[x].digitalSignals[digOffset+87].GoodQual;

		(* Reserve Signal 9 *)
		bPlaceHolderCustomSignal[x] 				:= IN_CU.tPlantCom_E2E_In_Cust10ms[x].digitalSignals[digOffset+88].Value;
		bPlaceHolderCustomSignalGoodQual[x] 		:= IN_CU.tPlantCom_E2E_In_Cust10ms[x].digitalSignals[digOffset+88].GoodQual;

		(* Reserve Signal 10 *)
		bPlaceHolderCustomSignal[x] 				:=	IN_CU.tPlantCom_E2E_In_Cust10ms[x].digitalSignals[digOffset+89].Value;
		bPlaceHolderCustomSignalGoodQual[x] 		:= IN_CU.tPlantCom_E2E_In_Cust10ms[x].digitalSignals[digOffset+89].GoodQual;

		(* Reserve Signal 11 *)
		bPlaceHolderCustomSignal[x] 				:= IN_CU.tPlantCom_E2E_In_Cust10ms[x].digitalSignals[digOffset+90].Value;
		bPlaceHolderCustomSignalGoodQual[x]			:= IN_CU.tPlantCom_E2E_In_Cust10ms[x].digitalSignals[digOffset+90].GoodQual;

		(* Reserve Signal 12 *)
		bPlaceHolderCustomSignal[x] 				:= IN_CU.tPlantCom_E2E_In_Cust10ms[x].digitalSignals[digOffset+91].Value;
		bPlaceHolderCustomSignalGoodQual[x] 		:= IN_CU.tPlantCom_E2E_In_Cust10ms[x].digitalSignals[digOffset+91].GoodQual;

		(* Reserve Signal 13 *)
		bPlaceHolderCustomSignal[x] 				:= IN_CU.tPlantCom_E2E_In_Cust10ms[x].digitalSignals[digOffset+92].Value;
		bPlaceHolderCustomSignalGoodQual[x] 		:= IN_CU.tPlantCom_E2E_In_Cust10ms[x].digitalSignals[digOffset+92].GoodQual;

		(* Reserve Signal 14 *)
		bPlaceHolderCustomSignal[x] 				:= IN_CU.tPlantCom_E2E_In_Cust10ms[x].digitalSignals[digOffset+93].Value;
		bPlaceHolderCustomSignalGoodQual[x] 		:= IN_CU.tPlantCom_E2E_In_Cust10ms[x].digitalSignals[digOffset+93].GoodQual;

		(* Reserve Signal 15 *)
		bPlaceHolderCustomSignal[x] 				:= IN_CU.tPlantCom_E2E_In_Cust10ms[x].digitalSignals[digOffset+94].Value;
		bPlaceHolderCustomSignalGoodQual[x] 		:= IN_CU.tPlantCom_E2E_In_Cust10ms[x].digitalSignals[digOffset+94].GoodQual;

		(* Reserve Signal 16 *)
		bPlaceHolderCustomSignal[x] 				:= IN_CU.tPlantCom_E2E_In_Cust10ms[x].digitalSignals[digOffset+95].Value;
		bPlaceHolderCustomSignalGoodQual[x] 		:= IN_CU.tPlantCom_E2E_In_Cust10ms[x].digitalSignals[digOffset+95].GoodQual;

		(**********************)
		(*** Analog Signals ***)
		(**********************)

		(* Reserve Signal 1 *)
		rPlaceHolderCustomSignal[x] 				:= IN_CU.tPlantCom_E2E_In_Cust10ms[x].analogSignals[anaOffset+40].Value;
		bPlaceHolderCustomSignalGoodQual[x] 		:= IN_CU.tPlantCom_E2E_In_Cust10ms[x].analogSignals[anaOffset+40].GoodQual;

		(* Reserve Signal 2 *)
		rPlaceHolderCustomSignal[x] 				:= IN_CU.tPlantCom_E2E_In_Cust10ms[x].analogSignals[anaOffset+41].Value;
		bPlaceHolderCustomSignalGoodQual[x]			:= IN_CU.tPlantCom_E2E_In_Cust10ms[x].analogSignals[anaOffset+41].GoodQual;

		(* Reserve Signal 3 *)
		rPlaceHolderCustomSignal[x] 				:= IN_CU.tPlantCom_E2E_In_Cust10ms[x].analogSignals[anaOffset+42].Value;
		bPlaceHolderCustomSignalGoodQual[x] 		:= IN_CU.tPlantCom_E2E_In_Cust10ms[x].analogSignals[anaOffset+42].GoodQual;

		(* Reserve Signal 4 *)
		rPlaceHolderCustomSignal[x] 				:= IN_CU.tPlantCom_E2E_In_Cust10ms[x].analogSignals[anaOffset+43].Value;
		bPlaceHolderCustomSignalGoodQual[x] 		:= IN_CU.tPlantCom_E2E_In_Cust10ms[x].analogSignals[anaOffset+43].GoodQual;

		(* Reserve Signal 5 *)
		rPlaceHolderCustomSignal[x] 				:= IN_CU.tPlantCom_E2E_In_Cust10ms[x].analogSignals[anaOffset+44].Value;
		bPlaceHolderCustomSignalGoodQual[x] 		:= IN_CU.tPlantCom_E2E_In_Cust10ms[x].analogSignals[anaOffset+44].GoodQual;

		(* Reserve Signal 6 *)
		rPlaceHolderCustomSignal[x] 				:= IN_CU.tPlantCom_E2E_In_Cust10ms[x].analogSignals[anaOffset+45].Value;
		bPlaceHolderCustomSignalGoodQual[x] 		:= IN_CU.tPlantCom_E2E_In_Cust10ms[x].analogSignals[anaOffset+45].GoodQual;

		(* Reserve Signal 7 *)
		rPlaceHolderCustomSignal[x] 				:= IN_CU.tPlantCom_E2E_In_Cust10ms[x].analogSignals[anaOffset+46].Value;
		bPlaceHolderCustomSignalGoodQual[x]			:= IN_CU.tPlantCom_E2E_In_Cust10ms[x].analogSignals[anaOffset+46].GoodQual;

		(* Reserve Signal 8 *)
		rPlaceHolderCustomSignal[x]					:= IN_CU.tPlantCom_E2E_In_Cust10ms[x].analogSignals[anaOffset+47].Value;
		bPlaceHolderCustomSignalGoodQual[x] 		:= IN_CU.tPlantCom_E2E_In_Cust10ms[x].analogSignals[anaOffset+47].GoodQual;
	END_FOR

	(*** Customized Outputs to the other engines ***)

	(***********************)
	(*** Digital Signals ***)
	(***********************)
	bPlaceHolderCustomSignal[0] := FALSE;
	(* Reserve Signal 1 *)
	OUT_CU.tPlantCom_E2E_Out_Cust10ms.digitalSignals[digOffset+80].Value 			:= bPlaceHolderCustomSignal[0];
	OUT_CU.tPlantCom_E2E_Out_Cust10ms.digitalSignals[digOffset+80].GoodQual 		:= TRUE;

	(* Reserve Signal 2 *)
	OUT_CU.tPlantCom_E2E_Out_Cust10ms.digitalSignals[digOffset+81].Value 			:= bPlaceHolderCustomSignal[0];
	OUT_CU.tPlantCom_E2E_Out_Cust10ms.digitalSignals[digOffset+81].GoodQual 		:= TRUE;

	(* Reserve Signal 3 *)
	OUT_CU.tPlantCom_E2E_Out_Cust10ms.digitalSignals[digOffset+82].Value 			:= bPlaceHolderCustomSignal[0];
	OUT_CU.tPlantCom_E2E_Out_Cust10ms.digitalSignals[digOffset+82].GoodQual 		:= TRUE;

	(* Reserve Signal 4 *)
	OUT_CU.tPlantCom_E2E_Out_Cust10ms.digitalSignals[digOffset+83].Value 			:= bPlaceHolderCustomSignal[0];
	OUT_CU.tPlantCom_E2E_Out_Cust10ms.digitalSignals[digOffset+83].GoodQual 		:= TRUE;

	(* Reserve Signal 5 *)
	OUT_CU.tPlantCom_E2E_Out_Cust10ms.digitalSignals[digOffset+84].Value 			:= bPlaceHolderCustomSignal[0];
	OUT_CU.tPlantCom_E2E_Out_Cust10ms.digitalSignals[digOffset+84].GoodQual 		:= TRUE;

	(* Reserve Signal 6 *)
	OUT_CU.tPlantCom_E2E_Out_Cust10ms.digitalSignals[digOffset+85].Value 			:= bPlaceHolderCustomSignal[0];
	OUT_CU.tPlantCom_E2E_Out_Cust10ms.digitalSignals[digOffset+85].GoodQual 		:= TRUE;

	(* Reserve Signal 7 *)
	OUT_CU.tPlantCom_E2E_Out_Cust10ms.digitalSignals[digOffset+86].Value 			:= bPlaceHolderCustomSignal[0];
	OUT_CU.tPlantCom_E2E_Out_Cust10ms.digitalSignals[digOffset+86].GoodQual 		:= TRUE;

	(* Reserve Signal 8 *)
	OUT_CU.tPlantCom_E2E_Out_Cust10ms.digitalSignals[digOffset+87].Value 			:= bPlaceHolderCustomSignal[0];
	OUT_CU.tPlantCom_E2E_Out_Cust10ms.digitalSignals[digOffset+87].GoodQual 		:= TRUE;

	(* Reserve Signal 9 *)
	OUT_CU.tPlantCom_E2E_Out_Cust10ms.digitalSignals[digOffset+88].Value 			:= bPlaceHolderCustomSignal[0];
	OUT_CU.tPlantCom_E2E_Out_Cust10ms.digitalSignals[digOffset+88].GoodQual 		:= TRUE;

	(* Reserve Signal 10 *)
	OUT_CU.tPlantCom_E2E_Out_Cust10ms.digitalSignals[digOffset+89].Value 			:= bPlaceHolderCustomSignal[0];
	OUT_CU.tPlantCom_E2E_Out_Cust10ms.digitalSignals[digOffset+89].GoodQual 		:= TRUE;

	(* Reserve Signal 11 *)
	OUT_CU.tPlantCom_E2E_Out_Cust10ms.digitalSignals[digOffset+90].Value 			:= bPlaceHolderCustomSignal[0];
	OUT_CU.tPlantCom_E2E_Out_Cust10ms.digitalSignals[digOffset+90].GoodQual 		:= TRUE;

	(* Reserve Signal 12 *)
	OUT_CU.tPlantCom_E2E_Out_Cust10ms.digitalSignals[digOffset+91].Value 			:= bPlaceHolderCustomSignal[0];
	OUT_CU.tPlantCom_E2E_Out_Cust10ms.digitalSignals[digOffset+91].GoodQual 		:= TRUE;

	(* Reserve Signal 13 *)
	OUT_CU.tPlantCom_E2E_Out_Cust10ms.digitalSignals[digOffset+92].Value 			:= bPlaceHolderCustomSignal[0];
	OUT_CU.tPlantCom_E2E_Out_Cust10ms.digitalSignals[digOffset+92].GoodQual 		:= TRUE;

	(* Reserve Signal 14 *)
	OUT_CU.tPlantCom_E2E_Out_Cust10ms.digitalSignals[digOffset+93].Value 			:= bPlaceHolderCustomSignal[0];
	OUT_CU.tPlantCom_E2E_Out_Cust10ms.digitalSignals[digOffset+93].GoodQual 		:= TRUE;

	(* Reserve Signal 15 *)
	OUT_CU.tPlantCom_E2E_Out_Cust10ms.digitalSignals[digOffset+94].Value 			:= bPlaceHolderCustomSignal[0];
	OUT_CU.tPlantCom_E2E_Out_Cust10ms.digitalSignals[digOffset+94].GoodQual 		:= TRUE;

	(* Reserve Signal 16 *)
	OUT_CU.tPlantCom_E2E_Out_Cust10ms.digitalSignals[digOffset+95].Value 			:= bPlaceHolderCustomSignal[0];
	OUT_CU.tPlantCom_E2E_Out_Cust10ms.digitalSignals[digOffset+95].GoodQual 		:= TRUE;

	(**********************)
	(*** Analog Signals ***)
	(**********************)
	rPlaceHolderCustomSignal[0] := 0.00;
	(* Reserve Signal 1 *)
	OUT_CU.tPlantCom_E2E_Out_Cust10ms.analogSignals[anaOffset+40].Value 			:= rPlaceHolderCustomSignal[0];
	OUT_CU.tPlantCom_E2E_Out_Cust10ms.analogSignals[anaOffset+40].GoodQual 			:= TRUE;

	(* Reserve Signal 2 *)
	OUT_CU.tPlantCom_E2E_Out_Cust10ms.analogSignals[anaOffset+41].Value 			:= rPlaceHolderCustomSignal[0];
	OUT_CU.tPlantCom_E2E_Out_Cust10ms.analogSignals[anaOffset+41].GoodQual 			:= TRUE;

	(* Reserve Signal 3 *)
	OUT_CU.tPlantCom_E2E_Out_Cust10ms.analogSignals[anaOffset+42].Value 			:= rPlaceHolderCustomSignal[0];
	OUT_CU.tPlantCom_E2E_Out_Cust10ms.analogSignals[anaOffset+42].GoodQual 			:= TRUE;

	(* Reserve Signal 4 *)
	OUT_CU.tPlantCom_E2E_Out_Cust10ms.analogSignals[anaOffset+43].Value 			:= rPlaceHolderCustomSignal[0];
	OUT_CU.tPlantCom_E2E_Out_Cust10ms.analogSignals[anaOffset+43].GoodQual 			:= TRUE;

	(* Reserve Signal 5 *)
	OUT_CU.tPlantCom_E2E_Out_Cust10ms.analogSignals[anaOffset+44].Value 			:= rPlaceHolderCustomSignal[0];
	OUT_CU.tPlantCom_E2E_Out_Cust10ms.analogSignals[anaOffset+44].GoodQual 			:= TRUE;

	(* Reserve Signal 6 *)
	OUT_CU.tPlantCom_E2E_Out_Cust10ms.analogSignals[anaOffset+45].Value 			:= rPlaceHolderCustomSignal[0];
	OUT_CU.tPlantCom_E2E_Out_Cust10ms.analogSignals[anaOffset+45].GoodQual 			:= TRUE;

	(* Reserve Signal 7 *)
	OUT_CU.tPlantCom_E2E_Out_Cust10ms.analogSignals[anaOffset+46].Value 			:= rPlaceHolderCustomSignal[0];
	OUT_CU.tPlantCom_E2E_Out_Cust10ms.analogSignals[anaOffset+46].GoodQual 			:= TRUE;

	(* Reserve Signal 8 *)
	OUT_CU.tPlantCom_E2E_Out_Cust10ms.analogSignals[anaOffset+47].Value 			:= rPlaceHolderCustomSignal[0];
	OUT_CU.tPlantCom_E2E_Out_Cust10ms.analogSignals[anaOffset+47].GoodQual 			:= TRUE;

END_PROGRAM
```

#### Init.st - Init code
```iecst
(*******************************************************************************
Customized Variable mapping for the plant communication

This code is confidential and proprietary to the INNIO Company.
It may not be used in any form, or reproduced in any manner, without the express
written permission of the INNIO Company.
Copyright, INNIO Company, 2024

Customized modifications: -
------------------------

History:
-------
V4.14.0	26.11.2024	Astner	Created Task

Instructions for use: -
--------------------
Outstandings: -
------------

*******************************************************************************)

PROGRAM _INIT
	(* Insert code here *)

END_PROGRAM
```

#### Variables.var - Local variables
```iecst
(*Helper Variables*)
VAR CONSTANT
	anaOffset : SINT := -40;
	digOffset : SINT := -80;
END_VAR
VAR
	x : USINT := 0;
	bPlaceHolderCustomSignal : ARRAY[0..32] OF BOOL := [33(FALSE)];
	rPlaceHolderCustomSignal : ARRAY[0..32] OF REAL := [33(0.0)];
	bPlaceHolderCustomSignalGoodQual : ARRAY[0..32] OF BOOL := [33(FALSE)];
END_VAR
```

### Program Logical/Customized/PlantCom/c_PlantComMap100ms (IEC, version 4.14.0)

#### Cyclic.st - Cyclic code
```iecst
(*******************************************************************************
Customized Variable mapping for the plant communication

This code is confidential and proprietary to the INNIO Company.
It may not be used in any form, or reproduced in any manner, without the express
written permission of the INNIO Company.
Copyright, INNIO Company, 2024

Customized modifications: -
------------------------

History:
-------
V4.14.0	26.11.2024	Astner	Created Task

Instructions for use:
--------------------
Replace the bPlaceholderCustomSignal[x] variable with the variable you want to add to the plant communication.
The GoodQual Value of the Output variables must be always true by default, if additional logic is needed this
has to be implemented in the software module where the variable is coming from.
The GoodQual Value of the inputs is set by the communication participant.
Outstandings:
------------

*******************************************************************************)
PROGRAM _CYCLIC
	(* Do not exeucte mapping if plant communication is not configured *)
	IF (NOT IN_CU.bPlantComCfgOk) THEN
		RETURN;
	END_IF

	(***************************************************)
	(*** Customized Inputs from the master controls  ***)
	(***************************************************)

	FOR x:=Para.tPlantComm.iMas_Num_Min TO Para.tPlantComm.iMas_Num_Max DO
		(***********************)
		(*** Digital Signals ***)
		(***********************)
		(* Reserve Signal 1 *)
		bPlaceHolderCustomSignal[x]             := IN_CU.tPlantCom_M2E_In_Cust100ms[x].digitalSignals[digOffset+32].Value;
		bPlaceHolderCustomSignalGoodQual[x]     := IN_CU.tPlantCom_M2E_In_Cust100ms[x].digitalSignals[digOffset+32].GoodQual;

		(* Reserve Signal 2 *)
		bPlaceHolderCustomSignal[x]             := IN_CU.tPlantCom_M2E_In_Cust100ms[x].digitalSignals[digOffset+33].Value;
		bPlaceHolderCustomSignalGoodQual[x]     := IN_CU.tPlantCom_M2E_In_Cust100ms[x].digitalSignals[digOffset+33].GoodQual;

		(* Reserve Signal 3 *)
		bPlaceHolderCustomSignal[x]             := IN_CU.tPlantCom_M2E_In_Cust100ms[x].digitalSignals[digOffset+34].Value;
		bPlaceHolderCustomSignalGoodQual[x]     := IN_CU.tPlantCom_M2E_In_Cust100ms[x].digitalSignals[digOffset+34].GoodQual;

		(* Reserve Signal 4 *)
		bPlaceHolderCustomSignal[x]             := IN_CU.tPlantCom_M2E_In_Cust100ms[x].digitalSignals[digOffset+35].Value;
		bPlaceHolderCustomSignalGoodQual[x]     := IN_CU.tPlantCom_M2E_In_Cust100ms[x].digitalSignals[digOffset+35].GoodQual;

		(* Reserve Signal 5 *)
		bPlaceHolderCustomSignal[x]             := IN_CU.tPlantCom_M2E_In_Cust100ms[x].digitalSignals[digOffset+36].Value;
		bPlaceHolderCustomSignalGoodQual[x]     := IN_CU.tPlantCom_M2E_In_Cust100ms[x].digitalSignals[digOffset+36].GoodQual;

		(* Reserve Signal 6 *)
		bPlaceHolderCustomSignal[x]             := IN_CU.tPlantCom_M2E_In_Cust100ms[x].digitalSignals[digOffset+37].Value;
		bPlaceHolderCustomSignalGoodQual[x]     := IN_CU.tPlantCom_M2E_In_Cust100ms[x].digitalSignals[digOffset+37].GoodQual;

		(* Reserve Signal 7 *)
		bPlaceHolderCustomSignal[x]             := IN_CU.tPlantCom_M2E_In_Cust100ms[x].digitalSignals[digOffset+38].Value;
		bPlaceHolderCustomSignalGoodQual[x]     := IN_CU.tPlantCom_M2E_In_Cust100ms[x].digitalSignals[digOffset+38].GoodQual;

		(* Reserve Signal 8 *)
		bPlaceHolderCustomSignal[x]             := IN_CU.tPlantCom_M2E_In_Cust100ms[x].digitalSignals[digOffset+39].Value;
		bPlaceHolderCustomSignalGoodQual[x]     := IN_CU.tPlantCom_M2E_In_Cust100ms[x].digitalSignals[digOffset+39].GoodQual;

		(* Reserve Signal 9 *)
		bPlaceHolderCustomSignal[x]             := IN_CU.tPlantCom_M2E_In_Cust100ms[x].digitalSignals[digOffset+40].Value;
		bPlaceHolderCustomSignalGoodQual[x]     := IN_CU.tPlantCom_M2E_In_Cust100ms[x].digitalSignals[digOffset+40].GoodQual;

		(* Reserve Signal 10 *)
		bPlaceHolderCustomSignal[x]             := IN_CU.tPlantCom_M2E_In_Cust100ms[x].digitalSignals[digOffset+41].Value;
		bPlaceHolderCustomSignalGoodQual[x]     := IN_CU.tPlantCom_M2E_In_Cust100ms[x].digitalSignals[digOffset+41].GoodQual;

		(* Reserve Signal 11 *)
		bPlaceHolderCustomSignal[x]             := IN_CU.tPlantCom_M2E_In_Cust100ms[x].digitalSignals[digOffset+42].Value;
		bPlaceHolderCustomSignalGoodQual[x]     := IN_CU.tPlantCom_M2E_In_Cust100ms[x].digitalSignals[digOffset+42].GoodQual;

		(* Reserve Signal 12 *)
		bPlaceHolderCustomSignal[x]             := IN_CU.tPlantCom_M2E_In_Cust100ms[x].digitalSignals[digOffset+43].Value;
		bPlaceHolderCustomSignalGoodQual[x]     := IN_CU.tPlantCom_M2E_In_Cust100ms[x].digitalSignals[digOffset+43].GoodQual;

		(* Reserve Signal 13 *)
		bPlaceHolderCustomSignal[x]             := IN_CU.tPlantCom_M2E_In_Cust100ms[x].digitalSignals[digOffset+44].Value;
		bPlaceHolderCustomSignalGoodQual[x]     := IN_CU.tPlantCom_M2E_In_Cust100ms[x].digitalSignals[digOffset+44].GoodQual;

		(* Reserve Signal 14 *)
		bPlaceHolderCustomSignal[x]             := IN_CU.tPlantCom_M2E_In_Cust100ms[x].digitalSignals[digOffset+45].Value;
		bPlaceHolderCustomSignalGoodQual[x]     := IN_CU.tPlantCom_M2E_In_Cust100ms[x].digitalSignals[digOffset+45].GoodQual;

		(* Reserve Signal 15 *)
		bPlaceHolderCustomSignal[x]             := IN_CU.tPlantCom_M2E_In_Cust100ms[x].digitalSignals[digOffset+46].Value;
		bPlaceHolderCustomSignalGoodQual[x]     := IN_CU.tPlantCom_M2E_In_Cust100ms[x].digitalSignals[digOffset+46].GoodQual;

		(* Reserve Signal 16 *)
		bPlaceHolderCustomSignal[x]             := IN_CU.tPlantCom_M2E_In_Cust100ms[x].digitalSignals[digOffset+47].Value;
		bPlaceHolderCustomSignalGoodQual[x]     := IN_CU.tPlantCom_M2E_In_Cust100ms[x].digitalSignals[digOffset+47].GoodQual;

		(* Reserve Signal 17 *)
		bPlaceHolderCustomSignal[x]             := IN_CU.tPlantCom_M2E_In_Cust100ms[x].digitalSignals[digOffset+48].Value;
		bPlaceHolderCustomSignalGoodQual[x]     := IN_CU.tPlantCom_M2E_In_Cust100ms[x].digitalSignals[digOffset+48].GoodQual;

		(* Reserve Signal 18 *)
		bPlaceHolderCustomSignal[x]             := IN_CU.tPlantCom_M2E_In_Cust100ms[x].digitalSignals[digOffset+49].Value;
		bPlaceHolderCustomSignalGoodQual[x]     := IN_CU.tPlantCom_M2E_In_Cust100ms[x].digitalSignals[digOffset+49].GoodQual;

		(* Reserve Signal 19 *)
		bPlaceHolderCustomSignal[x]             := IN_CU.tPlantCom_M2E_In_Cust100ms[x].digitalSignals[digOffset+50].Value;
		bPlaceHolderCustomSignalGoodQual[x]     := IN_CU.tPlantCom_M2E_In_Cust100ms[x].digitalSignals[digOffset+50].GoodQual;

		(* Reserve Signal 20 *)
		bPlaceHolderCustomSignal[x]             := IN_CU.tPlantCom_M2E_In_Cust100ms[x].digitalSignals[digOffset+51].Value;
		bPlaceHolderCustomSignalGoodQual[x]     := IN_CU.tPlantCom_M2E_In_Cust100ms[x].digitalSignals[digOffset+51].GoodQual;

		(* Reserve Signal 21 *)
		bPlaceHolderCustomSignal[x]             := IN_CU.tPlantCom_M2E_In_Cust100ms[x].digitalSignals[digOffset+52].Value;
		bPlaceHolderCustomSignalGoodQual[x]     := IN_CU.tPlantCom_M2E_In_Cust100ms[x].digitalSignals[digOffset+52].GoodQual;

		(* Reserve Signal 22 *)
		bPlaceHolderCustomSignal[x]             := IN_CU.tPlantCom_M2E_In_Cust100ms[x].digitalSignals[digOffset+53].Value;
		bPlaceHolderCustomSignalGoodQual[x]     := IN_CU.tPlantCom_M2E_In_Cust100ms[x].digitalSignals[digOffset+53].GoodQual;

		(* Reserve Signal 23 *)
		bPlaceHolderCustomSignal[x]             := IN_CU.tPlantCom_M2E_In_Cust100ms[x].digitalSignals[digOffset+54].Value;
		bPlaceHolderCustomSignalGoodQual[x]     := IN_CU.tPlantCom_M2E_In_Cust100ms[x].digitalSignals[digOffset+54].GoodQual;

		(* Reserve Signal 24 *)
		bPlaceHolderCustomSignal[x]             := IN_CU.tPlantCom_M2E_In_Cust100ms[x].digitalSignals[digOffset+55].Value;
		bPlaceHolderCustomSignalGoodQual[x]     := IN_CU.tPlantCom_M2E_In_Cust100ms[x].digitalSignals[digOffset+55].GoodQual;

		(* Reserve Signal 25 *)
		bPlaceHolderCustomSignal[x]             := IN_CU.tPlantCom_M2E_In_Cust100ms[x].digitalSignals[digOffset+56].Value;
		bPlaceHolderCustomSignalGoodQual[x]     := IN_CU.tPlantCom_M2E_In_Cust100ms[x].digitalSignals[digOffset+56].GoodQual;

		(* Reserve Signal 26 *)
		bPlaceHolderCustomSignal[x]             := IN_CU.tPlantCom_M2E_In_Cust100ms[x].digitalSignals[digOffset+57].Value;
		bPlaceHolderCustomSignalGoodQual[x]     := IN_CU.tPlantCom_M2E_In_Cust100ms[x].digitalSignals[digOffset+57].GoodQual;

		(* Reserve Signal 27 *)
		bPlaceHolderCustomSignal[x]             := IN_CU.tPlantCom_M2E_In_Cust100ms[x].digitalSignals[digOffset+58].Value;
		bPlaceHolderCustomSignalGoodQual[x]     := IN_CU.tPlantCom_M2E_In_Cust100ms[x].digitalSignals[digOffset+58].GoodQual;

		(* Reserve Signal 28 *)
		bPlaceHolderCustomSignal[x]             := IN_CU.tPlantCom_M2E_In_Cust100ms[x].digitalSignals[digOffset+59].Value;
		bPlaceHolderCustomSignalGoodQual[x]     := IN_CU.tPlantCom_M2E_In_Cust100ms[x].digitalSignals[digOffset+59].GoodQual;

		(* Reserve Signal 29 *)
		bPlaceHolderCustomSignal[x]             := IN_CU.tPlantCom_M2E_In_Cust100ms[x].digitalSignals[digOffset+60].Value;
		bPlaceHolderCustomSignalGoodQual[x]     := IN_CU.tPlantCom_M2E_In_Cust100ms[x].digitalSignals[digOffset+60].GoodQual;

		(* Reserve Signal 30 *)
		bPlaceHolderCustomSignal[x]             := IN_CU.tPlantCom_M2E_In_Cust100ms[x].digitalSignals[digOffset+61].Value;
		bPlaceHolderCustomSignalGoodQual[x]     := IN_CU.tPlantCom_M2E_In_Cust100ms[x].digitalSignals[digOffset+61].GoodQual;

		(* Reserve Signal 31 *)
		bPlaceHolderCustomSignal[x]             := IN_CU.tPlantCom_M2E_In_Cust100ms[x].digitalSignals[digOffset+62].Value;
		bPlaceHolderCustomSignalGoodQual[x]     := IN_CU.tPlantCom_M2E_In_Cust100ms[x].digitalSignals[digOffset+62].GoodQual;

		(* Reserve Signal 32 *)
		bPlaceHolderCustomSignal[x]             := IN_CU.tPlantCom_M2E_In_Cust100ms[x].digitalSignals[digOffset+63].Value;
		bPlaceHolderCustomSignalGoodQual[x]     := IN_CU.tPlantCom_M2E_In_Cust100ms[x].digitalSignals[digOffset+63].GoodQual;

		(**********************)
		(*** Analog Signals ***)
		(**********************)

		(* Reserve Signal 1 *)
		rPlaceHolderCustomSignal[x]             := IN_CU.tPlantCom_M2E_In_Cust100ms[x].analogSignals[anaOffset+16].Value;
		bPlaceHolderCustomSignalGoodQual[x]     := IN_CU.tPlantCom_M2E_In_Cust100ms[x].analogSignals[anaOffset+16].GoodQual;

		(* Reserve Signal 2 *)
		rPlaceHolderCustomSignal[x]             := IN_CU.tPlantCom_M2E_In_Cust100ms[x].analogSignals[anaOffset+17].Value;
		bPlaceHolderCustomSignalGoodQual[x]     := IN_CU.tPlantCom_M2E_In_Cust100ms[x].analogSignals[anaOffset+17].GoodQual;

		(* Reserve Signal 3 *)
		rPlaceHolderCustomSignal[x]             := IN_CU.tPlantCom_M2E_In_Cust100ms[x].analogSignals[anaOffset+18].Value;
		bPlaceHolderCustomSignalGoodQual[x]     := IN_CU.tPlantCom_M2E_In_Cust100ms[x].analogSignals[anaOffset+18].GoodQual;

		(* Reserve Signal 4 *)
		rPlaceHolderCustomSignal[x]             := IN_CU.tPlantCom_M2E_In_Cust100ms[x].analogSignals[anaOffset+19].Value;
		bPlaceHolderCustomSignalGoodQual[x]     := IN_CU.tPlantCom_M2E_In_Cust100ms[x].analogSignals[anaOffset+19].GoodQual;

		(* Reserve Signal 5 *)
		rPlaceHolderCustomSignal[x]             := IN_CU.tPlantCom_M2E_In_Cust100ms[x].analogSignals[anaOffset+20].Value;
		bPlaceHolderCustomSignalGoodQual[x]     := IN_CU.tPlantCom_M2E_In_Cust100ms[x].analogSignals[anaOffset+20].GoodQual;

		(* Reserve Signal 6 *)
		rPlaceHolderCustomSignal[x]             := IN_CU.tPlantCom_M2E_In_Cust100ms[x].analogSignals[anaOffset+21].Value;
		bPlaceHolderCustomSignalGoodQual[x]     := IN_CU.tPlantCom_M2E_In_Cust100ms[x].analogSignals[anaOffset+21].GoodQual;

		(* Reserve Signal 7 *)
		rPlaceHolderCustomSignal[x]             := IN_CU.tPlantCom_M2E_In_Cust100ms[x].analogSignals[anaOffset+22].Value;
		bPlaceHolderCustomSignalGoodQual[x]     := IN_CU.tPlantCom_M2E_In_Cust100ms[x].analogSignals[anaOffset+22].GoodQual;

		(* Reserve Signal 8 *)
		rPlaceHolderCustomSignal[x]             := IN_CU.tPlantCom_M2E_In_Cust100ms[x].analogSignals[anaOffset+23].Value;
		bPlaceHolderCustomSignalGoodQual[x]     := IN_CU.tPlantCom_M2E_In_Cust100ms[x].analogSignals[anaOffset+23].GoodQual;

		(* Reserve Signal 9 *)
		rPlaceHolderCustomSignal[x]             := IN_CU.tPlantCom_M2E_In_Cust100ms[x].analogSignals[anaOffset+24].Value;
		bPlaceHolderCustomSignalGoodQual[x]     := IN_CU.tPlantCom_M2E_In_Cust100ms[x].analogSignals[anaOffset+24].GoodQual;

		(* Reserve Signal 10 *)
		rPlaceHolderCustomSignal[x]             := IN_CU.tPlantCom_M2E_In_Cust100ms[x].analogSignals[anaOffset+25].Value;
		bPlaceHolderCustomSignalGoodQual[x]     := IN_CU.tPlantCom_M2E_In_Cust100ms[x].analogSignals[anaOffset+25].GoodQual;

		(* Reserve Signal 11 *)
		rPlaceHolderCustomSignal[x]             := IN_CU.tPlantCom_M2E_In_Cust100ms[x].analogSignals[anaOffset+26].Value;
		bPlaceHolderCustomSignalGoodQual[x]     := IN_CU.tPlantCom_M2E_In_Cust100ms[x].analogSignals[anaOffset+26].GoodQual;

		(* Reserve Signal 12 *)
		rPlaceHolderCustomSignal[x]             := IN_CU.tPlantCom_M2E_In_Cust100ms[x].analogSignals[anaOffset+27].Value;
		bPlaceHolderCustomSignalGoodQual[x]     := IN_CU.tPlantCom_M2E_In_Cust100ms[x].analogSignals[anaOffset+27].GoodQual;

		(* Reserve Signal 13 *)
		rPlaceHolderCustomSignal[x]             := IN_CU.tPlantCom_M2E_In_Cust100ms[x].analogSignals[anaOffset+28].Value;
		bPlaceHolderCustomSignalGoodQual[x]     := IN_CU.tPlantCom_M2E_In_Cust100ms[x].analogSignals[anaOffset+28].GoodQual;

		(* Reserve Signal 14 *)
		rPlaceHolderCustomSignal[x]             := IN_CU.tPlantCom_M2E_In_Cust100ms[x].analogSignals[anaOffset+29].Value;
		bPlaceHolderCustomSignalGoodQual[x]     := IN_CU.tPlantCom_M2E_In_Cust100ms[x].analogSignals[anaOffset+29].GoodQual;

		(* Reserve Signal 15 *)
		rPlaceHolderCustomSignal[x]             := IN_CU.tPlantCom_M2E_In_Cust100ms[x].analogSignals[anaOffset+30].Value;
		bPlaceHolderCustomSignalGoodQual[x]     := IN_CU.tPlantCom_M2E_In_Cust100ms[x].analogSignals[anaOffset+30].GoodQual;

		(* Reserve Signal 16 *)
		rPlaceHolderCustomSignal[x]             := IN_CU.tPlantCom_M2E_In_Cust100ms[x].analogSignals[anaOffset+31].Value;
		bPlaceHolderCustomSignalGoodQual[x]     := IN_CU.tPlantCom_M2E_In_Cust100ms[x].analogSignals[anaOffset+31].GoodQual;
	END_FOR

	(*** Customized Outputs to the master controls  ***)
	FOR x:=Para.tPlantComm.iMas_Num_Min TO Para.tPlantComm.iMas_Num_Max DO
		(***********************)
		(*** Digital Signals ***)
		(***********************)
		bPlaceHolderCustomSignal[x] := FALSE;
		(* Reserve Signal 1 *)
		OUT_CU.tPlantCom_E2M_Out_Cust100ms[x].digitalSignals[digOffset+32].Value          := bPlaceHolderCustomSignal[x];
		OUT_CU.tPlantCom_E2M_Out_Cust100ms[x].digitalSignals[digOffset+32].GoodQual       := TRUE;

		(* Reserve Signal 2 *)
		OUT_CU.tPlantCom_E2M_Out_Cust100ms[x].digitalSignals[digOffset+33].Value          := bPlaceHolderCustomSignal[x];
		OUT_CU.tPlantCom_E2M_Out_Cust100ms[x].digitalSignals[digOffset+33].GoodQual       := TRUE;

		(* Reserve Signal 3 *)
		OUT_CU.tPlantCom_E2M_Out_Cust100ms[x].digitalSignals[digOffset+34].Value          := bPlaceHolderCustomSignal[x];
		OUT_CU.tPlantCom_E2M_Out_Cust100ms[x].digitalSignals[digOffset+34].GoodQual       := TRUE;

		(* Reserve Signal 4 *)
		OUT_CU.tPlantCom_E2M_Out_Cust100ms[x].digitalSignals[digOffset+35].Value          := bPlaceHolderCustomSignal[x];
		OUT_CU.tPlantCom_E2M_Out_Cust100ms[x].digitalSignals[digOffset+35].GoodQual       := TRUE;

		(* Reserve Signal 5 *)
		OUT_CU.tPlantCom_E2M_Out_Cust100ms[x].digitalSignals[digOffset+36].Value          := bPlaceHolderCustomSignal[x];
		OUT_CU.tPlantCom_E2M_Out_Cust100ms[x].digitalSignals[digOffset+36].GoodQual       := TRUE;

		(* Reserve Signal 6 *)
		OUT_CU.tPlantCom_E2M_Out_Cust100ms[x].digitalSignals[digOffset+37].Value          := bPlaceHolderCustomSignal[x];
		OUT_CU.tPlantCom_E2M_Out_Cust100ms[x].digitalSignals[digOffset+37].GoodQual       := TRUE;

		(* Reserve Signal 7 *)
		OUT_CU.tPlantCom_E2M_Out_Cust100ms[x].digitalSignals[digOffset+38].Value          := bPlaceHolderCustomSignal[x];
		OUT_CU.tPlantCom_E2M_Out_Cust100ms[x].digitalSignals[digOffset+38].GoodQual       := TRUE;

		(* Reserve Signal 8 *)
		OUT_CU.tPlantCom_E2M_Out_Cust100ms[x].digitalSignals[digOffset+39].Value          := bPlaceHolderCustomSignal[x];
		OUT_CU.tPlantCom_E2M_Out_Cust100ms[x].digitalSignals[digOffset+39].GoodQual       := TRUE;

		(* Reserve Signal 9 *)
		OUT_CU.tPlantCom_E2M_Out_Cust100ms[x].digitalSignals[digOffset+40].Value          := bPlaceHolderCustomSignal[x];
		OUT_CU.tPlantCom_E2M_Out_Cust100ms[x].digitalSignals[digOffset+40].GoodQual       := TRUE;

		(* Reserve Signal 10 *)
		OUT_CU.tPlantCom_E2M_Out_Cust100ms[x].digitalSignals[digOffset+41].Value          := bPlaceHolderCustomSignal[x];
		OUT_CU.tPlantCom_E2M_Out_Cust100ms[x].digitalSignals[digOffset+41].GoodQual       := TRUE;

		(* Reserve Signal 11 *)
		OUT_CU.tPlantCom_E2M_Out_Cust100ms[x].digitalSignals[digOffset+42].Value          := bPlaceHolderCustomSignal[x];
		OUT_CU.tPlantCom_E2M_Out_Cust100ms[x].digitalSignals[digOffset+42].GoodQual       := TRUE;

		(* Reserve Signal 12 *)
		OUT_CU.tPlantCom_E2M_Out_Cust100ms[x].digitalSignals[digOffset+43].Value          := bPlaceHolderCustomSignal[x];
		OUT_CU.tPlantCom_E2M_Out_Cust100ms[x].digitalSignals[digOffset+43].GoodQual       := TRUE;

		(* Reserve Signal 13 *)
		OUT_CU.tPlantCom_E2M_Out_Cust100ms[x].digitalSignals[digOffset+44].Value          := bPlaceHolderCustomSignal[x];
		OUT_CU.tPlantCom_E2M_Out_Cust100ms[x].digitalSignals[digOffset+44].GoodQual       := TRUE;

		(* Reserve Signal 14 *)
		OUT_CU.tPlantCom_E2M_Out_Cust100ms[x].digitalSignals[digOffset+45].Value          := bPlaceHolderCustomSignal[x];
		OUT_CU.tPlantCom_E2M_Out_Cust100ms[x].digitalSignals[digOffset+45].GoodQual       := TRUE;

		(* Reserve Signal 15 *)
		OUT_CU.tPlantCom_E2M_Out_Cust100ms[x].digitalSignals[digOffset+46].Value          := bPlaceHolderCustomSignal[x];
		OUT_CU.tPlantCom_E2M_Out_Cust100ms[x].digitalSignals[digOffset+46].GoodQual       := TRUE;

		(* Reserve Signal 16 *)
		OUT_CU.tPlantCom_E2M_Out_Cust100ms[x].digitalSignals[digOffset+47].Value          := bPlaceHolderCustomSignal[x];
		OUT_CU.tPlantCom_E2M_Out_Cust100ms[x].digitalSignals[digOffset+47].GoodQual       := TRUE;

		(* Reserve Signal 17 *)
		OUT_CU.tPlantCom_E2M_Out_Cust100ms[x].digitalSignals[digOffset+48].Value          := bPlaceHolderCustomSignal[x];
		OUT_CU.tPlantCom_E2M_Out_Cust100ms[x].digitalSignals[digOffset+48].GoodQual       := TRUE;

		(* Reserve Signal 18 *)
		OUT_CU.tPlantCom_E2M_Out_Cust100ms[x].digitalSignals[digOffset+49].Value          := bPlaceHolderCustomSignal[x];
		OUT_CU.tPlantCom_E2M_Out_Cust100ms[x].digitalSignals[digOffset+49].GoodQual       := TRUE;

		(* Reserve Signal 19 *)
		OUT_CU.tPlantCom_E2M_Out_Cust100ms[x].digitalSignals[digOffset+50].Value          := bPlaceHolderCustomSignal[x];
		OUT_CU.tPlantCom_E2M_Out_Cust100ms[x].digitalSignals[digOffset+50].GoodQual       := TRUE;

		(* Reserve Signal 20 *)
		OUT_CU.tPlantCom_E2M_Out_Cust100ms[x].digitalSignals[digOffset+51].Value          := bPlaceHolderCustomSignal[x];
		OUT_CU.tPlantCom_E2M_Out_Cust100ms[x].digitalSignals[digOffset+51].GoodQual       := TRUE;

		(* Reserve Signal 21 *)
		OUT_CU.tPlantCom_E2M_Out_Cust100ms[x].digitalSignals[digOffset+52].Value          := bPlaceHolderCustomSignal[x];
		OUT_CU.tPlantCom_E2M_Out_Cust100ms[x].digitalSignals[digOffset+52].GoodQual       := TRUE;

		(* Reserve Signal 22 *)
		OUT_CU.tPlantCom_E2M_Out_Cust100ms[x].digitalSignals[digOffset+53].Value          := bPlaceHolderCustomSignal[x];
		OUT_CU.tPlantCom_E2M_Out_Cust100ms[x].digitalSignals[digOffset+53].GoodQual       := TRUE;

		(* Reserve Signal 23 *)
		OUT_CU.tPlantCom_E2M_Out_Cust100ms[x].digitalSignals[digOffset+54].Value          := bPlaceHolderCustomSignal[x];
		OUT_CU.tPlantCom_E2M_Out_Cust100ms[x].digitalSignals[digOffset+54].GoodQual       := TRUE;

		(* Reserve Signal 24 *)
		OUT_CU.tPlantCom_E2M_Out_Cust100ms[x].digitalSignals[digOffset+55].Value          := bPlaceHolderCustomSignal[x];
		OUT_CU.tPlantCom_E2M_Out_Cust100ms[x].digitalSignals[digOffset+55].GoodQual       := TRUE;

		(* Reserve Signal 25 *)
		OUT_CU.tPlantCom_E2M_Out_Cust100ms[x].digitalSignals[digOffset+56].Value          := bPlaceHolderCustomSignal[x];
		OUT_CU.tPlantCom_E2M_Out_Cust100ms[x].digitalSignals[digOffset+56].GoodQual       := TRUE;

		(* Reserve Signal 26 *)
		OUT_CU.tPlantCom_E2M_Out_Cust100ms[x].digitalSignals[digOffset+57].Value          := bPlaceHolderCustomSignal[x];
		OUT_CU.tPlantCom_E2M_Out_Cust100ms[x].digitalSignals[digOffset+57].GoodQual       := TRUE;

		(* Reserve Signal 27 *)
		OUT_CU.tPlantCom_E2M_Out_Cust100ms[x].digitalSignals[digOffset+58].Value          := bPlaceHolderCustomSignal[x];
		OUT_CU.tPlantCom_E2M_Out_Cust100ms[x].digitalSignals[digOffset+58].GoodQual       := TRUE;

		(* Reserve Signal 28 *)
		OUT_CU.tPlantCom_E2M_Out_Cust100ms[x].digitalSignals[digOffset+59].Value          := bPlaceHolderCustomSignal[x];
		OUT_CU.tPlantCom_E2M_Out_Cust100ms[x].digitalSignals[digOffset+59].GoodQual       := TRUE;

		(* Reserve Signal 29 *)
		OUT_CU.tPlantCom_E2M_Out_Cust100ms[x].digitalSignals[digOffset+60].Value          := bPlaceHolderCustomSignal[x];
		OUT_CU.tPlantCom_E2M_Out_Cust100ms[x].digitalSignals[digOffset+60].GoodQual       := TRUE;

		(* Reserve Signal 30 *)
		OUT_CU.tPlantCom_E2M_Out_Cust100ms[x].digitalSignals[digOffset+61].Value          := bPlaceHolderCustomSignal[x];
		OUT_CU.tPlantCom_E2M_Out_Cust100ms[x].digitalSignals[digOffset+61].GoodQual       := TRUE;

		(* Reserve Signal 31 *)
		OUT_CU.tPlantCom_E2M_Out_Cust100ms[x].digitalSignals[digOffset+62].Value          := bPlaceHolderCustomSignal[x];
		OUT_CU.tPlantCom_E2M_Out_Cust100ms[x].digitalSignals[digOffset+62].GoodQual       := TRUE;

		(* Reserve Signal 32 *)
		OUT_CU.tPlantCom_E2M_Out_Cust100ms[x].digitalSignals[digOffset+63].Value          := bPlaceHolderCustomSignal[x];
		OUT_CU.tPlantCom_E2M_Out_Cust100ms[x].digitalSignals[digOffset+63].GoodQual       := TRUE;

		(**********************)
		(*** Analog Signals ***)
		(**********************)
		rPlaceHolderCustomSignal[x] := 0.0;
		(* Reserve Signal 1 *)
		OUT_CU.tPlantCom_E2M_Out_Cust100ms[x].analogSignals[anaOffset+16].Value          := rPlaceHolderCustomSignal[x];
		OUT_CU.tPlantCom_E2M_Out_Cust100ms[x].analogSignals[anaOffset+16].GoodQual       := TRUE;

		(* Reserve Signal 2 *)
		OUT_CU.tPlantCom_E2M_Out_Cust100ms[x].analogSignals[anaOffset+17].Value          := rPlaceHolderCustomSignal[x];
		OUT_CU.tPlantCom_E2M_Out_Cust100ms[x].analogSignals[anaOffset+17].GoodQual       := TRUE;

		(* Reserve Signal 3 *)
		OUT_CU.tPlantCom_E2M_Out_Cust100ms[x].analogSignals[anaOffset+18].Value          := rPlaceHolderCustomSignal[x];
		OUT_CU.tPlantCom_E2M_Out_Cust100ms[x].analogSignals[anaOffset+18].GoodQual       := TRUE;

		(* Reserve Signal 4 *)
		OUT_CU.tPlantCom_E2M_Out_Cust100ms[x].analogSignals[anaOffset+19].Value          := rPlaceHolderCustomSignal[x];
		OUT_CU.tPlantCom_E2M_Out_Cust100ms[x].analogSignals[anaOffset+19].GoodQual       := TRUE;

		(* Reserve Signal 5 *)
		OUT_CU.tPlantCom_E2M_Out_Cust100ms[x].analogSignals[anaOffset+20].Value          := rPlaceHolderCustomSignal[x];
		OUT_CU.tPlantCom_E2M_Out_Cust100ms[x].analogSignals[anaOffset+20].GoodQual       := TRUE;

		(* Reserve Signal 6 *)
		OUT_CU.tPlantCom_E2M_Out_Cust100ms[x].analogSignals[anaOffset+21].Value          := rPlaceHolderCustomSignal[x];
		OUT_CU.tPlantCom_E2M_Out_Cust100ms[x].analogSignals[anaOffset+21].GoodQual       := TRUE;

		(* Reserve Signal 7 *)
		OUT_CU.tPlantCom_E2M_Out_Cust100ms[x].analogSignals[anaOffset+22].Value          := rPlaceHolderCustomSignal[x];
		OUT_CU.tPlantCom_E2M_Out_Cust100ms[x].analogSignals[anaOffset+22].GoodQual       := TRUE;

		(* Reserve Signal 8 *)
		OUT_CU.tPlantCom_E2M_Out_Cust100ms[x].analogSignals[anaOffset+23].Value          := rPlaceHolderCustomSignal[x];
		OUT_CU.tPlantCom_E2M_Out_Cust100ms[x].analogSignals[anaOffset+23].GoodQual       := TRUE;

		(* Reserve Signal 9 *)
		OUT_CU.tPlantCom_E2M_Out_Cust100ms[x].analogSignals[anaOffset+24].Value          := rPlaceHolderCustomSignal[x];
		OUT_CU.tPlantCom_E2M_Out_Cust100ms[x].analogSignals[anaOffset+24].GoodQual       := TRUE;

		(* Reserve Signal 10 *)
		OUT_CU.tPlantCom_E2M_Out_Cust100ms[x].analogSignals[anaOffset+25].Value          := rPlaceHolderCustomSignal[x];
		OUT_CU.tPlantCom_E2M_Out_Cust100ms[x].analogSignals[anaOffset+25].GoodQual       := TRUE;

		(* Reserve Signal 11 *)
		OUT_CU.tPlantCom_E2M_Out_Cust100ms[x].analogSignals[anaOffset+26].Value          := rPlaceHolderCustomSignal[x];
		OUT_CU.tPlantCom_E2M_Out_Cust100ms[x].analogSignals[anaOffset+26].GoodQual       := TRUE;

		(* Reserve Signal 12 *)
		OUT_CU.tPlantCom_E2M_Out_Cust100ms[x].analogSignals[anaOffset+27].Value          := rPlaceHolderCustomSignal[x];
		OUT_CU.tPlantCom_E2M_Out_Cust100ms[x].analogSignals[anaOffset+27].GoodQual       := TRUE;

		(* Reserve Signal 13 *)
		OUT_CU.tPlantCom_E2M_Out_Cust100ms[x].analogSignals[anaOffset+28].Value          := rPlaceHolderCustomSignal[x];
		OUT_CU.tPlantCom_E2M_Out_Cust100ms[x].analogSignals[anaOffset+28].GoodQual       := TRUE;

		(* Reserve Signal 14 *)
		OUT_CU.tPlantCom_E2M_Out_Cust100ms[x].analogSignals[anaOffset+29].Value          := rPlaceHolderCustomSignal[x];
		OUT_CU.tPlantCom_E2M_Out_Cust100ms[x].analogSignals[anaOffset+29].GoodQual       := TRUE;

		(* Reserve Signal 15 *)
		OUT_CU.tPlantCom_E2M_Out_Cust100ms[x].analogSignals[anaOffset+30].Value          := rPlaceHolderCustomSignal[x];
		OUT_CU.tPlantCom_E2M_Out_Cust100ms[x].analogSignals[anaOffset+30].GoodQual       := TRUE;

		(* Reserve Signal 16 *)
		OUT_CU.tPlantCom_E2M_Out_Cust100ms[x].analogSignals[anaOffset+31].Value          := rPlaceHolderCustomSignal[x];
		OUT_CU.tPlantCom_E2M_Out_Cust100ms[x].analogSignals[anaOffset+31].GoodQual       := TRUE;
	END_FOR

	(*** Customized Inputs from the other engines ***)
	FOR x:=Para.tPlantComm.iEng_Num_Min TO Para.tPlantComm.iEng_Num_Max DO
		(***********************)
		(*** Digital Signals ***)
		(***********************)

		(* Reserve Signal 1 *)
		bPlaceHolderCustomSignal[x]                     := IN_CU.tPlantCom_E2E_In_Cust100ms[x].digitalSignals[digOffset+32].Value;
		bPlaceHolderCustomSignalGoodQual[x]             := IN_CU.tPlantCom_E2E_In_Cust100ms[x].digitalSignals[digOffset+32].GoodQual;

		(* Reserve Signal 2 *)
		bPlaceHolderCustomSignal[x]                     := IN_CU.tPlantCom_E2E_In_Cust100ms[x].digitalSignals[digOffset+33].Value;
		bPlaceHolderCustomSignalGoodQual[x]             := IN_CU.tPlantCom_E2E_In_Cust100ms[x].digitalSignals[digOffset+33].GoodQual;

		(* Reserve Signal 3 *)
		bPlaceHolderCustomSignal[x]                     := IN_CU.tPlantCom_E2E_In_Cust100ms[x].digitalSignals[digOffset+34].Value;
		bPlaceHolderCustomSignalGoodQual[x]             := IN_CU.tPlantCom_E2E_In_Cust100ms[x].digitalSignals[digOffset+34].GoodQual;

		(* Reserve Signal 4 *)
		bPlaceHolderCustomSignal[x]                     := IN_CU.tPlantCom_E2E_In_Cust100ms[x].digitalSignals[digOffset+35].Value;
		bPlaceHolderCustomSignalGoodQual[x]             := IN_CU.tPlantCom_E2E_In_Cust100ms[x].digitalSignals[digOffset+35].GoodQual;

		(* Reserve Signal 5 *)
		bPlaceHolderCustomSignal[x]                     := IN_CU.tPlantCom_E2E_In_Cust100ms[x].digitalSignals[digOffset+36].Value;
		bPlaceHolderCustomSignalGoodQual[x]             := IN_CU.tPlantCom_E2E_In_Cust100ms[x].digitalSignals[digOffset+36].GoodQual;

		(* Reserve Signal 6 *)
		bPlaceHolderCustomSignal[x]                     := IN_CU.tPlantCom_E2E_In_Cust100ms[x].digitalSignals[digOffset+37].Value;
		bPlaceHolderCustomSignalGoodQual[x]             := IN_CU.tPlantCom_E2E_In_Cust100ms[x].digitalSignals[digOffset+37].GoodQual;

		(* Reserve Signal 7 *)
		bPlaceHolderCustomSignal[x]                     := IN_CU.tPlantCom_E2E_In_Cust100ms[x].digitalSignals[digOffset+38].Value;
		bPlaceHolderCustomSignalGoodQual[x]             := IN_CU.tPlantCom_E2E_In_Cust100ms[x].digitalSignals[digOffset+38].GoodQual;

		(* Reserve Signal 8 *)
		bPlaceHolderCustomSignal[x]                     := IN_CU.tPlantCom_E2E_In_Cust100ms[x].digitalSignals[digOffset+39].Value;
		bPlaceHolderCustomSignalGoodQual[x]             := IN_CU.tPlantCom_E2E_In_Cust100ms[x].digitalSignals[digOffset+39].GoodQual;

		(* Reserve Signal 9 *)
		bPlaceHolderCustomSignal[x]                     := IN_CU.tPlantCom_E2E_In_Cust100ms[x].digitalSignals[digOffset+40].Value;
		bPlaceHolderCustomSignalGoodQual[x]             := IN_CU.tPlantCom_E2E_In_Cust100ms[x].digitalSignals[digOffset+40].GoodQual;

		(* Reserve Signal 10 *)
		bPlaceHolderCustomSignal[x]                     := IN_CU.tPlantCom_E2E_In_Cust100ms[x].digitalSignals[digOffset+41].Value;
		bPlaceHolderCustomSignalGoodQual[x]             := IN_CU.tPlantCom_E2E_In_Cust100ms[x].digitalSignals[digOffset+41].GoodQual;

		(* Reserve Signal 11 *)
		bPlaceHolderCustomSignal[x]                     := IN_CU.tPlantCom_E2E_In_Cust100ms[x].digitalSignals[digOffset+42].Value;
		bPlaceHolderCustomSignalGoodQual[x]             := IN_CU.tPlantCom_E2E_In_Cust100ms[x].digitalSignals[digOffset+42].GoodQual;

		(* Reserve Signal 12 *)
		bPlaceHolderCustomSignal[x]                     := IN_CU.tPlantCom_E2E_In_Cust100ms[x].digitalSignals[digOffset+43].Value;
		bPlaceHolderCustomSignalGoodQual[x]             := IN_CU.tPlantCom_E2E_In_Cust100ms[x].digitalSignals[digOffset+43].GoodQual;

		(* Reserve Signal 13 *)
		bPlaceHolderCustomSignal[x]                     := IN_CU.tPlantCom_E2E_In_Cust100ms[x].digitalSignals[digOffset+44].Value;
		bPlaceHolderCustomSignalGoodQual[x]             := IN_CU.tPlantCom_E2E_In_Cust100ms[x].digitalSignals[digOffset+44].GoodQual;

		(* Reserve Signal 14 *)
		bPlaceHolderCustomSignal[x]                     := IN_CU.tPlantCom_E2E_In_Cust100ms[x].digitalSignals[digOffset+45].Value;
		bPlaceHolderCustomSignalGoodQual[x]             := IN_CU.tPlantCom_E2E_In_Cust100ms[x].digitalSignals[digOffset+45].GoodQual;

		(* Reserve Signal 15 *)
		bPlaceHolderCustomSignal[x]                     := IN_CU.tPlantCom_E2E_In_Cust100ms[x].digitalSignals[digOffset+46].Value;
		bPlaceHolderCustomSignalGoodQual[x]             := IN_CU.tPlantCom_E2E_In_Cust100ms[x].digitalSignals[digOffset+46].GoodQual;

		(* Reserve Signal 16 *)
		bPlaceHolderCustomSignal[x]                     := IN_CU.tPlantCom_E2E_In_Cust100ms[x].digitalSignals[digOffset+47].Value;
		bPlaceHolderCustomSignalGoodQual[x]             := IN_CU.tPlantCom_E2E_In_Cust100ms[x].digitalSignals[digOffset+47].GoodQual;

		(* Reserve Signal 17 *)
		bPlaceHolderCustomSignal[x]                     := IN_CU.tPlantCom_E2E_In_Cust100ms[x].digitalSignals[digOffset+48].Value;
		bPlaceHolderCustomSignalGoodQual[x]             := IN_CU.tPlantCom_E2E_In_Cust100ms[x].digitalSignals[digOffset+48].GoodQual;

		(* Reserve Signal 18 *)
		bPlaceHolderCustomSignal[x]                     := IN_CU.tPlantCom_E2E_In_Cust100ms[x].digitalSignals[digOffset+49].Value;
		bPlaceHolderCustomSignalGoodQual[x]             := IN_CU.tPlantCom_E2E_In_Cust100ms[x].digitalSignals[digOffset+49].GoodQual;

		(* Reserve Signal 19 *)
		bPlaceHolderCustomSignal[x]                     := IN_CU.tPlantCom_E2E_In_Cust100ms[x].digitalSignals[digOffset+50].Value;
		bPlaceHolderCustomSignalGoodQual[x]             := IN_CU.tPlantCom_E2E_In_Cust100ms[x].digitalSignals[digOffset+50].GoodQual;

		(* Reserve Signal 20 *)
		bPlaceHolderCustomSignal[x]                     := IN_CU.tPlantCom_E2E_In_Cust100ms[x].digitalSignals[digOffset+51].Value;
		bPlaceHolderCustomSignalGoodQual[x]             := IN_CU.tPlantCom_E2E_In_Cust100ms[x].digitalSignals[digOffset+51].GoodQual;

		(* Reserve Signal 21 *)
		bPlaceHolderCustomSignal[x]                     := IN_CU.tPlantCom_E2E_In_Cust100ms[x].digitalSignals[digOffset+52].Value;
		bPlaceHolderCustomSignalGoodQual[x]             := IN_CU.tPlantCom_E2E_In_Cust100ms[x].digitalSignals[digOffset+52].GoodQual;

		(* Reserve Signal 22 *)
		bPlaceHolderCustomSignal[x]                     := IN_CU.tPlantCom_E2E_In_Cust100ms[x].digitalSignals[digOffset+53].Value;
		bPlaceHolderCustomSignalGoodQual[x]             := IN_CU.tPlantCom_E2E_In_Cust100ms[x].digitalSignals[digOffset+53].GoodQual;

		(* Reserve Signal 23 *)
		bPlaceHolderCustomSignal[x]                     := IN_CU.tPlantCom_E2E_In_Cust100ms[x].digitalSignals[digOffset+54].Value;
		bPlaceHolderCustomSignalGoodQual[x]             := IN_CU.tPlantCom_E2E_In_Cust100ms[x].digitalSignals[digOffset+54].GoodQual;

		(* Reserve Signal 24 *)
		bPlaceHolderCustomSignal[x]                     := IN_CU.tPlantCom_E2E_In_Cust100ms[x].digitalSignals[digOffset+55].Value;
		bPlaceHolderCustomSignalGoodQual[x]             := IN_CU.tPlantCom_E2E_In_Cust100ms[x].digitalSignals[digOffset+55].GoodQual;

		(* Reserve Signal 25 *)
		bPlaceHolderCustomSignal[x]                     := IN_CU.tPlantCom_E2E_In_Cust100ms[x].digitalSignals[digOffset+56].Value;
		bPlaceHolderCustomSignalGoodQual[x]             := IN_CU.tPlantCom_E2E_In_Cust100ms[x].digitalSignals[digOffset+56].GoodQual;

		(* Reserve Signal 26 *)
		bPlaceHolderCustomSignal[x]                     := IN_CU.tPlantCom_E2E_In_Cust100ms[x].digitalSignals[digOffset+57].Value;
		bPlaceHolderCustomSignalGoodQual[x]             := IN_CU.tPlantCom_E2E_In_Cust100ms[x].digitalSignals[digOffset+57].GoodQual;

		(* Reserve Signal 27 *)
		bPlaceHolderCustomSignal[x]                     := IN_CU.tPlantCom_E2E_In_Cust100ms[x].digitalSignals[digOffset+58].Value;
		bPlaceHolderCustomSignalGoodQual[x]             := IN_CU.tPlantCom_E2E_In_Cust100ms[x].digitalSignals[digOffset+58].GoodQual;

		(* Reserve Signal 28 *)
		bPlaceHolderCustomSignal[x]                     := IN_CU.tPlantCom_E2E_In_Cust100ms[x].digitalSignals[digOffset+59].Value;
		bPlaceHolderCustomSignalGoodQual[x]             := IN_CU.tPlantCom_E2E_In_Cust100ms[x].digitalSignals[digOffset+59].GoodQual;

		(* Reserve Signal 29 *)
		bPlaceHolderCustomSignal[x]                     := IN_CU.tPlantCom_E2E_In_Cust100ms[x].digitalSignals[digOffset+60].Value;
		bPlaceHolderCustomSignalGoodQual[x]             := IN_CU.tPlantCom_E2E_In_Cust100ms[x].digitalSignals[digOffset+60].GoodQual;

		(* Reserve Signal 30 *)
		bPlaceHolderCustomSignal[x]                     := IN_CU.tPlantCom_E2E_In_Cust100ms[x].digitalSignals[digOffset+61].Value;
		bPlaceHolderCustomSignalGoodQual[x]             := IN_CU.tPlantCom_E2E_In_Cust100ms[x].digitalSignals[digOffset+61].GoodQual;

		(* Reserve Signal 31 *)
		bPlaceHolderCustomSignal[x]                     := IN_CU.tPlantCom_E2E_In_Cust100ms[x].digitalSignals[digOffset+62].Value;
		bPlaceHolderCustomSignalGoodQual[x]             := IN_CU.tPlantCom_E2E_In_Cust100ms[x].digitalSignals[digOffset+62].GoodQual;

		(* Reserve Signal 32 *)
		bPlaceHolderCustomSignal[x]                     := IN_CU.tPlantCom_E2E_In_Cust100ms[x].digitalSignals[digOffset+63].Value;
		bPlaceHolderCustomSignalGoodQual[x]             := IN_CU.tPlantCom_E2E_In_Cust100ms[x].digitalSignals[digOffset+63].GoodQual;

		(**********************)
		(*** Analog Signals ***)
		(**********************)

		(* Reserve Signal 1 *)
		rPlaceHolderCustomSignal[x]                     := IN_CU.tPlantCom_E2E_In_Cust100ms[x].analogSignals[anaOffset+16].Value;
		bPlaceHolderCustomSignalGoodQual[x]             := IN_CU.tPlantCom_E2E_In_Cust100ms[x].analogSignals[anaOffset+16].GoodQual;

		(* Reserve Signal 2 *)
		rPlaceHolderCustomSignal[x]                     := IN_CU.tPlantCom_E2E_In_Cust100ms[x].analogSignals[anaOffset+17].Value;
		bPlaceHolderCustomSignalGoodQual[x]             := IN_CU.tPlantCom_E2E_In_Cust100ms[x].analogSignals[anaOffset+17].GoodQual;

		(* Reserve Signal 3 *)
		rPlaceHolderCustomSignal[x]                     := IN_CU.tPlantCom_E2E_In_Cust100ms[x].analogSignals[anaOffset+18].Value;
		bPlaceHolderCustomSignalGoodQual[x]             := IN_CU.tPlantCom_E2E_In_Cust100ms[x].analogSignals[anaOffset+18].GoodQual;

		(* Reserve Signal 4 *)
		rPlaceHolderCustomSignal[x]                     := IN_CU.tPlantCom_E2E_In_Cust100ms[x].analogSignals[anaOffset+19].Value;
		bPlaceHolderCustomSignalGoodQual[x]             := IN_CU.tPlantCom_E2E_In_Cust100ms[x].analogSignals[anaOffset+19].GoodQual;

		(* Reserve Signal 5 *)
		rPlaceHolderCustomSignal[x]                     := IN_CU.tPlantCom_E2E_In_Cust100ms[x].analogSignals[anaOffset+20].Value;
		bPlaceHolderCustomSignalGoodQual[x]             := IN_CU.tPlantCom_E2E_In_Cust100ms[x].analogSignals[anaOffset+20].GoodQual;

		(* Reserve Signal 6 *)
		rPlaceHolderCustomSignal[x]                     := IN_CU.tPlantCom_E2E_In_Cust100ms[x].analogSignals[anaOffset+21].Value;
		bPlaceHolderCustomSignalGoodQual[x]             := IN_CU.tPlantCom_E2E_In_Cust100ms[x].analogSignals[anaOffset+21].GoodQual;

		(* Reserve Signal 7 *)
		rPlaceHolderCustomSignal[x]                     := IN_CU.tPlantCom_E2E_In_Cust100ms[x].analogSignals[anaOffset+22].Value;
		bPlaceHolderCustomSignalGoodQual[x]             := IN_CU.tPlantCom_E2E_In_Cust100ms[x].analogSignals[anaOffset+22].GoodQual;

		(* Reserve Signal 8 *)
		rPlaceHolderCustomSignal[x]                     := IN_CU.tPlantCom_E2E_In_Cust100ms[x].analogSignals[anaOffset+23].Value;
		bPlaceHolderCustomSignalGoodQual[x]             := IN_CU.tPlantCom_E2E_In_Cust100ms[x].analogSignals[anaOffset+23].GoodQual;

		(* Reserve Signal 9 *)
		rPlaceHolderCustomSignal[x]                     := IN_CU.tPlantCom_E2E_In_Cust100ms[x].analogSignals[anaOffset+24].Value;
		bPlaceHolderCustomSignalGoodQual[x]             := IN_CU.tPlantCom_E2E_In_Cust100ms[x].analogSignals[anaOffset+24].GoodQual;

		(* Reserve Signal 10 *)
		rPlaceHolderCustomSignal[x]                     := IN_CU.tPlantCom_E2E_In_Cust100ms[x].analogSignals[anaOffset+25].Value;
		bPlaceHolderCustomSignalGoodQual[x]             := IN_CU.tPlantCom_E2E_In_Cust100ms[x].analogSignals[anaOffset+25].GoodQual;

		(* Reserve Signal 11 *)
		rPlaceHolderCustomSignal[x]                     := IN_CU.tPlantCom_E2E_In_Cust100ms[x].analogSignals[anaOffset+26].Value;
		bPlaceHolderCustomSignalGoodQual[x]             := IN_CU.tPlantCom_E2E_In_Cust100ms[x].analogSignals[anaOffset+26].GoodQual;

		(* Reserve Signal 12 *)
		rPlaceHolderCustomSignal[x]                     := IN_CU.tPlantCom_E2E_In_Cust100ms[x].analogSignals[anaOffset+27].Value;
		bPlaceHolderCustomSignalGoodQual[x]             := IN_CU.tPlantCom_E2E_In_Cust100ms[x].analogSignals[anaOffset+27].GoodQual;

		(* Reserve Signal 13 *)
		rPlaceHolderCustomSignal[x]                     := IN_CU.tPlantCom_E2E_In_Cust100ms[x].analogSignals[anaOffset+28].Value;
		bPlaceHolderCustomSignalGoodQual[x]             := IN_CU.tPlantCom_E2E_In_Cust100ms[x].analogSignals[anaOffset+28].GoodQual;

		(* Reserve Signal 14 *)
		rPlaceHolderCustomSignal[x]                     := IN_CU.tPlantCom_E2E_In_Cust100ms[x].analogSignals[anaOffset+29].Value;
		bPlaceHolderCustomSignalGoodQual[x]             := IN_CU.tPlantCom_E2E_In_Cust100ms[x].analogSignals[anaOffset+29].GoodQual;

		(* Reserve Signal 15 *)
		rPlaceHolderCustomSignal[x]                     := IN_CU.tPlantCom_E2E_In_Cust100ms[x].analogSignals[anaOffset+30].Value;
		bPlaceHolderCustomSignalGoodQual[x]             := IN_CU.tPlantCom_E2E_In_Cust100ms[x].analogSignals[anaOffset+30].GoodQual;

		(* Reserve Signal 16 *)
		rPlaceHolderCustomSignal[x]                     := IN_CU.tPlantCom_E2E_In_Cust100ms[x].analogSignals[anaOffset+31].Value;
		bPlaceHolderCustomSignalGoodQual[x]             := IN_CU.tPlantCom_E2E_In_Cust100ms[x].analogSignals[anaOffset+31].GoodQual;
	END_FOR

	(*** Customized Outputs to the other engines ***)

	(***********************)
	(*** Digital Signals ***)
	(***********************)
	bPlaceHolderCustomSignal[0] := FALSE;

	(* Reserve Signal 1 *)
	OUT_CU.tPlantCom_E2E_Out_Cust100ms.digitalSignals[digOffset+32].Value 			:= bPlaceHolderCustomSignal[0];
	OUT_CU.tPlantCom_E2E_Out_Cust100ms.digitalSignals[digOffset+32].GoodQual 		:= TRUE;

	(* Reserve Signal 2 *)
	OUT_CU.tPlantCom_E2E_Out_Cust100ms.digitalSignals[digOffset+33].Value 			:= bPlaceHolderCustomSignal[0];
	OUT_CU.tPlantCom_E2E_Out_Cust100ms.digitalSignals[digOffset+33].GoodQual 		:= TRUE;

	(* Reserve Signal 3 *)
	OUT_CU.tPlantCom_E2E_Out_Cust100ms.digitalSignals[digOffset+34].Value 			:= bPlaceHolderCustomSignal[0];
	OUT_CU.tPlantCom_E2E_Out_Cust100ms.digitalSignals[digOffset+34].GoodQual 		:= TRUE;

	(* Reserve Signal 4 *)
	OUT_CU.tPlantCom_E2E_Out_Cust100ms.digitalSignals[digOffset+35].Value 			:= bPlaceHolderCustomSignal[0];
	OUT_CU.tPlantCom_E2E_Out_Cust100ms.digitalSignals[digOffset+35].GoodQual 		:= TRUE;

	(* Reserve Signal 5 *)
	OUT_CU.tPlantCom_E2E_Out_Cust100ms.digitalSignals[digOffset+36].Value 			:= bPlaceHolderCustomSignal[0];
	OUT_CU.tPlantCom_E2E_Out_Cust100ms.digitalSignals[digOffset+36].GoodQual 		:= TRUE;

	(* Reserve Signal 6 *)
	OUT_CU.tPlantCom_E2E_Out_Cust100ms.digitalSignals[digOffset+37].Value 			:= bPlaceHolderCustomSignal[0];
	OUT_CU.tPlantCom_E2E_Out_Cust100ms.digitalSignals[digOffset+37].GoodQual 		:= TRUE;

	(* Reserve Signal 7 *)
	OUT_CU.tPlantCom_E2E_Out_Cust100ms.digitalSignals[digOffset+38].Value 			:= bPlaceHolderCustomSignal[0];
	OUT_CU.tPlantCom_E2E_Out_Cust100ms.digitalSignals[digOffset+38].GoodQual 		:= TRUE;

	(* Reserve Signal 8 *)
	OUT_CU.tPlantCom_E2E_Out_Cust100ms.digitalSignals[digOffset+39].Value 			:= bPlaceHolderCustomSignal[0];
	OUT_CU.tPlantCom_E2E_Out_Cust100ms.digitalSignals[digOffset+39].GoodQual 		:= TRUE;

	(* Reserve Signal 9 *)
	OUT_CU.tPlantCom_E2E_Out_Cust100ms.digitalSignals[digOffset+40].Value 			:= bPlaceHolderCustomSignal[0];
	OUT_CU.tPlantCom_E2E_Out_Cust100ms.digitalSignals[digOffset+40].GoodQual 		:= TRUE;

	(* Reserve Signal 10 *)
	OUT_CU.tPlantCom_E2E_Out_Cust100ms.digitalSignals[digOffset+41].Value 			:= bPlaceHolderCustomSignal[0];
	OUT_CU.tPlantCom_E2E_Out_Cust100ms.digitalSignals[digOffset+41].GoodQual 		:= TRUE;

	(* Reserve Signal 11 *)
	OUT_CU.tPlantCom_E2E_Out_Cust100ms.digitalSignals[digOffset+42].Value 			:= bPlaceHolderCustomSignal[0];
	OUT_CU.tPlantCom_E2E_Out_Cust100ms.digitalSignals[digOffset+42].GoodQual 		:= TRUE;

	(* Reserve Signal 12 *)
	OUT_CU.tPlantCom_E2E_Out_Cust100ms.digitalSignals[digOffset+43].Value 			:= bPlaceHolderCustomSignal[0];
	OUT_CU.tPlantCom_E2E_Out_Cust100ms.digitalSignals[digOffset+43].GoodQual 		:= TRUE;

	(* Reserve Signal 13 *)
	OUT_CU.tPlantCom_E2E_Out_Cust100ms.digitalSignals[digOffset+44].Value 			:= bPlaceHolderCustomSignal[0];
	OUT_CU.tPlantCom_E2E_Out_Cust100ms.digitalSignals[digOffset+44].GoodQual 		:= TRUE;

	(* Reserve Signal 14 *)
	OUT_CU.tPlantCom_E2E_Out_Cust100ms.digitalSignals[digOffset+45].Value 			:= bPlaceHolderCustomSignal[0];
	OUT_CU.tPlantCom_E2E_Out_Cust100ms.digitalSignals[digOffset+45].GoodQual 		:= TRUE;

	(* Reserve Signal 15 *)
	OUT_CU.tPlantCom_E2E_Out_Cust100ms.digitalSignals[digOffset+46].Value 			:= bPlaceHolderCustomSignal[0];
	OUT_CU.tPlantCom_E2E_Out_Cust100ms.digitalSignals[digOffset+46].GoodQual 		:= TRUE;

	(* Reserve Signal 16 *)
	OUT_CU.tPlantCom_E2E_Out_Cust100ms.digitalSignals[digOffset+47].Value 			:= bPlaceHolderCustomSignal[0];
	OUT_CU.tPlantCom_E2E_Out_Cust100ms.digitalSignals[digOffset+47].GoodQual 		:= TRUE;

	(* Reserve Signal 17 *)
	OUT_CU.tPlantCom_E2E_Out_Cust100ms.digitalSignals[digOffset+48].Value 			:= bPlaceHolderCustomSignal[0];
	OUT_CU.tPlantCom_E2E_Out_Cust100ms.digitalSignals[digOffset+48].GoodQual 		:= TRUE;

	(* Reserve Signal 18 *)
	OUT_CU.tPlantCom_E2E_Out_Cust100ms.digitalSignals[digOffset+49].Value 			:= bPlaceHolderCustomSignal[0];
	OUT_CU.tPlantCom_E2E_Out_Cust100ms.digitalSignals[digOffset+49].GoodQual 		:= TRUE;

	(* Reserve Signal 19 *)
	OUT_CU.tPlantCom_E2E_Out_Cust100ms.digitalSignals[digOffset+50].Value 			:= bPlaceHolderCustomSignal[0];
	OUT_CU.tPlantCom_E2E_Out_Cust100ms.digitalSignals[digOffset+50].GoodQual 		:= TRUE;

	(* Reserve Signal 20 *)
	OUT_CU.tPlantCom_E2E_Out_Cust100ms.digitalSignals[digOffset+51].Value 			:= bPlaceHolderCustomSignal[0];
	OUT_CU.tPlantCom_E2E_Out_Cust100ms.digitalSignals[digOffset+51].GoodQual 		:= TRUE;

	(* Reserve Signal 21 *)
	OUT_CU.tPlantCom_E2E_Out_Cust100ms.digitalSignals[digOffset+52].Value 			:= bPlaceHolderCustomSignal[0];
	OUT_CU.tPlantCom_E2E_Out_Cust100ms.digitalSignals[digOffset+52].GoodQual 		:= TRUE;

	(* Reserve Signal 22 *)
	OUT_CU.tPlantCom_E2E_Out_Cust100ms.digitalSignals[digOffset+53].Value 			:= bPlaceHolderCustomSignal[0];
	OUT_CU.tPlantCom_E2E_Out_Cust100ms.digitalSignals[digOffset+53].GoodQual 		:= TRUE;

	(* Reserve Signal 23 *)
	OUT_CU.tPlantCom_E2E_Out_Cust100ms.digitalSignals[digOffset+54].Value 			:= bPlaceHolderCustomSignal[0];
	OUT_CU.tPlantCom_E2E_Out_Cust100ms.digitalSignals[digOffset+54].GoodQual 		:= TRUE;

	(* Reserve Signal 24 *)
	OUT_CU.tPlantCom_E2E_Out_Cust100ms.digitalSignals[digOffset+55].Value 			:= bPlaceHolderCustomSignal[0];
	OUT_CU.tPlantCom_E2E_Out_Cust100ms.digitalSignals[digOffset+55].GoodQual 		:= TRUE;

	(* Reserve Signal 25 *)
	OUT_CU.tPlantCom_E2E_Out_Cust100ms.digitalSignals[digOffset+56].Value 			:= bPlaceHolderCustomSignal[0];
	OUT_CU.tPlantCom_E2E_Out_Cust100ms.digitalSignals[digOffset+56].GoodQual 		:= TRUE;

	(* Reserve Signal 26 *)
	OUT_CU.tPlantCom_E2E_Out_Cust100ms.digitalSignals[digOffset+57].Value 			:= bPlaceHolderCustomSignal[0];
	OUT_CU.tPlantCom_E2E_Out_Cust100ms.digitalSignals[digOffset+57].GoodQual 		:= TRUE;

	(* Reserve Signal 27 *)
	OUT_CU.tPlantCom_E2E_Out_Cust100ms.digitalSignals[digOffset+58].Value 			:= bPlaceHolderCustomSignal[0];
	OUT_CU.tPlantCom_E2E_Out_Cust100ms.digitalSignals[digOffset+58].GoodQual 		:= TRUE;

	(* Reserve Signal 28 *)
	OUT_CU.tPlantCom_E2E_Out_Cust100ms.digitalSignals[digOffset+59].Value 			:= bPlaceHolderCustomSignal[0];
	OUT_CU.tPlantCom_E2E_Out_Cust100ms.digitalSignals[digOffset+59].GoodQual 		:= TRUE;

	(* Reserve Signal 29 *)
	OUT_CU.tPlantCom_E2E_Out_Cust100ms.digitalSignals[digOffset+60].Value 			:= bPlaceHolderCustomSignal[0];
	OUT_CU.tPlantCom_E2E_Out_Cust100ms.digitalSignals[digOffset+60].GoodQual 		:= TRUE;

	(* Reserve Signal 30 *)
	OUT_CU.tPlantCom_E2E_Out_Cust100ms.digitalSignals[digOffset+61].Value 			:= bPlaceHolderCustomSignal[0];
	OUT_CU.tPlantCom_E2E_Out_Cust100ms.digitalSignals[digOffset+61].GoodQual 		:= TRUE;

	(* Reserve Signal 31 *)
	OUT_CU.tPlantCom_E2E_Out_Cust100ms.digitalSignals[digOffset+62].Value 			:= bPlaceHolderCustomSignal[0];
	OUT_CU.tPlantCom_E2E_Out_Cust100ms.digitalSignals[digOffset+62].GoodQual 		:= TRUE;

	(* Reserve Signal 32 *)
	OUT_CU.tPlantCom_E2E_Out_Cust100ms.digitalSignals[digOffset+63].Value 			:= bPlaceHolderCustomSignal[0];
	OUT_CU.tPlantCom_E2E_Out_Cust100ms.digitalSignals[digOffset+63].GoodQual 		:= TRUE;

	(**********************)
	(*** Analog Signals ***)
	(**********************)

	rPlaceHolderCustomSignal[0] := 0.0;

	(* Reserve Signal 1 *)
	OUT_CU.tPlantCom_E2E_Out_Cust100ms.analogSignals[anaOffset+16].Value 			:= rPlaceHolderCustomSignal[0];
	OUT_CU.tPlantCom_E2E_Out_Cust100ms.analogSignals[anaOffset+16].GoodQual 		:= TRUE;

	(* Reserve Signal 2 *)
	OUT_CU.tPlantCom_E2E_Out_Cust100ms.analogSignals[anaOffset+17].Value 			:= rPlaceHolderCustomSignal[0];
	OUT_CU.tPlantCom_E2E_Out_Cust100ms.analogSignals[anaOffset+17].GoodQual 		:= TRUE;

	(* Reserve Signal 3 *)
	OUT_CU.tPlantCom_E2E_Out_Cust100ms.analogSignals[anaOffset+18].Value 			:= rPlaceHolderCustomSignal[0];
	OUT_CU.tPlantCom_E2E_Out_Cust100ms.analogSignals[anaOffset+18].GoodQual 		:= TRUE;

	(* Reserve Signal 4 *)
	OUT_CU.tPlantCom_E2E_Out_Cust100ms.analogSignals[anaOffset+19].Value 			:= rPlaceHolderCustomSignal[0];
	OUT_CU.tPlantCom_E2E_Out_Cust100ms.analogSignals[anaOffset+19].GoodQual 		:= TRUE;

	(* Reserve Signal 5 *)
	OUT_CU.tPlantCom_E2E_Out_Cust100ms.analogSignals[anaOffset+20].Value 			:= rPlaceHolderCustomSignal[0];
	OUT_CU.tPlantCom_E2E_Out_Cust100ms.analogSignals[anaOffset+20].GoodQual 		:= TRUE;

	(* Reserve Signal 6 *)
	OUT_CU.tPlantCom_E2E_Out_Cust100ms.analogSignals[anaOffset+21].Value 			:= rPlaceHolderCustomSignal[0];
	OUT_CU.tPlantCom_E2E_Out_Cust100ms.analogSignals[anaOffset+21].GoodQual 		:= TRUE;

	(* Reserve Signal 7 *)
	OUT_CU.tPlantCom_E2E_Out_Cust100ms.analogSignals[anaOffset+22].Value 			:= rPlaceHolderCustomSignal[0];
	OUT_CU.tPlantCom_E2E_Out_Cust100ms.analogSignals[anaOffset+22].GoodQual 		:= TRUE;

	(* Reserve Signal 8 *)
	OUT_CU.tPlantCom_E2E_Out_Cust100ms.analogSignals[anaOffset+23].Value 			:= rPlaceHolderCustomSignal[0];
	OUT_CU.tPlantCom_E2E_Out_Cust100ms.analogSignals[anaOffset+23].GoodQual 		:= TRUE;

	(* Reserve Signal 9 *)
	OUT_CU.tPlantCom_E2E_Out_Cust100ms.analogSignals[anaOffset+24].Value 			:= rPlaceHolderCustomSignal[0];
	OUT_CU.tPlantCom_E2E_Out_Cust100ms.analogSignals[anaOffset+24].GoodQual 		:= TRUE;

	(* Reserve Signal 10 *)
	OUT_CU.tPlantCom_E2E_Out_Cust100ms.analogSignals[anaOffset+25].Value 			:= rPlaceHolderCustomSignal[0];
	OUT_CU.tPlantCom_E2E_Out_Cust100ms.analogSignals[anaOffset+25].GoodQual 		:= TRUE;

	(* Reserve Signal 11 *)
	OUT_CU.tPlantCom_E2E_Out_Cust100ms.analogSignals[anaOffset+26].Value 			:= rPlaceHolderCustomSignal[0];
	OUT_CU.tPlantCom_E2E_Out_Cust100ms.analogSignals[anaOffset+26].GoodQual 		:= TRUE;

	(* Reserve Signal 12 *)
	OUT_CU.tPlantCom_E2E_Out_Cust100ms.analogSignals[anaOffset+27].Value 			:= rPlaceHolderCustomSignal[0];
	OUT_CU.tPlantCom_E2E_Out_Cust100ms.analogSignals[anaOffset+27].GoodQual 		:= TRUE;

	(* Reserve Signal 13 *)
	OUT_CU.tPlantCom_E2E_Out_Cust100ms.analogSignals[anaOffset+28].Value 			:= rPlaceHolderCustomSignal[0];
	OUT_CU.tPlantCom_E2E_Out_Cust100ms.analogSignals[anaOffset+28].GoodQual 		:= TRUE;
	(* Reserve Signal 14 *)
	OUT_CU.tPlantCom_E2E_Out_Cust100ms.analogSignals[anaOffset+29].Value 			:= rPlaceHolderCustomSignal[0];
	OUT_CU.tPlantCom_E2E_Out_Cust100ms.analogSignals[anaOffset+29].GoodQual 		:= TRUE;

	(* Reserve Signal 15 *)
	OUT_CU.tPlantCom_E2E_Out_Cust100ms.analogSignals[anaOffset+30].Value 			:= rPlaceHolderCustomSignal[0];
	OUT_CU.tPlantCom_E2E_Out_Cust100ms.analogSignals[anaOffset+30].GoodQual 		:= TRUE;
	(* Reserve Signal 16 *)
	OUT_CU.tPlantCom_E2E_Out_Cust100ms.analogSignals[anaOffset+31].Value 			:= rPlaceHolderCustomSignal[0];
	OUT_CU.tPlantCom_E2E_Out_Cust100ms.analogSignals[anaOffset+31].GoodQual 		:= TRUE;

END_PROGRAM
```

#### Init.st - Init code
```iecst
(*******************************************************************************
Customized Variable mapping for the plant communication

This code is confidential and proprietary to the INNIO Company.
It may not be used in any form, or reproduced in any manner, without the express
written permission of the INNIO Company.
Copyright, INNIO Company, 2024

Customized modifications: -
------------------------

History:
-------
V4.14.0	26.11.2024	Astner	Created Task

Instructions for use: -
--------------------
Outstandings: -
------------

*******************************************************************************)

PROGRAM _INIT
	(* Insert code here *)

END_PROGRAM
```

#### Variables.var - Local variables
```iecst
(*Helper Variables*)
VAR CONSTANT
	digOffset : SINT := -32;
	anaOffset : SINT := -16;
END_VAR
VAR
	x : USINT := 0;
	bPlaceHolderCustomSignal : ARRAY[0..32] OF BOOL := [33(FALSE)];
	rPlaceHolderCustomSignal : ARRAY[0..32] OF REAL := [33(0.0)];
	bPlaceHolderCustomSignalGoodQual : ARRAY[0..32] OF BOOL := [33(FALSE)];
END_VAR
```

### Program Logical/Customized/c_clutch_CAN (IEC) - Horton CAN devices - J1939 protocol data read
